// TIA Portal project "PKS_projektna_naloga_v1_9" (V15.1)

(* hardware
DEVICE "S7-1200 station_1"  S7-1200 Station
   slot 0: "Rack_0"  S7-1200 Rack  Rack  V1.0
   slot 1: "PLC_1"  CPU 1214C DC/DC/DC  6ES7 214-1AG40-0XB0  V4.2
DEVICE "HMI_1"  TP700 Comfort
   slot 0: "HMI_1"  TP700 Comfort  6AV2 124-0GC01-0AX0  15.1.0.0
   slot 1: "HMI_RT_1"  TP700 Comfort  6AV2 124-0GC01-0AX0  15.1.0.0
   slot 5: "HMI_1.IE_CP_1"  PROFINET Interface  15.0.1.0
      slot 1: "PROFINET Interface_1"  PROFINET Interface
         slot 1: "Port_1"  Port
         slot 2: "Port_2"  Port
   slot 7: "HMI_1.MPI/DP_CP_1"  MPI/DP Interface  15.0.1.0
*)

// ===== PLC "PLC_1"  CPU 1214C DC/DC/DC =====
// protected blocks, not shown: "FB_sim_model"

VAR_GLOBAL   // PLC tag table "Default tag table"
   "Tag_1" AT %MD0 : Time;
   "Tag_2" AT %M0.0 : Bool;
END_VAR

DATA_BLOCK "DB_podatki_procesa"   // DB2
{ S7_Optimized_Access := 'TRUE' }
VERSION : 0.1
   VAR
      V_žel : Real := 3000.0;   // želeni volumen v posodi v ml
      mr_AB_žel : Real := 0.35;   // želeno mešalno razmerje (mA : mB)
      ventil_A_pretok_max : Real := 200.0;   // max pretok ventila v ml/s
      ventil_B_pretok : Real := 200.0;   // pretok ventila B v g/s
      m_posode : Real := 200.0;   // masa (prazne) posode v g
      čas_prekinitve : Real := 0.1;   // čas prekinitve v s
      t_žel_meš : Real := 10.0;   // želeni čas postopka mešanja v s
      t_žel_vib : Real := 5.0;   // želeni čas postopka na vibracijski plošči v s
   END_VAR
   VAR RETAIN
      init_pogoj : Bool;   // pogoj za inicializacijo spremenljivk
   END_VAR
BEGIN
END_DATA_BLOCK

DATA_BLOCK "DB_spremenljivke"   // DB3
{ S7_Optimized_Access := 'TRUE' }
VERSION : 0.1
   VAR
      glavno_stikalo : Bool;   // glavno stikalo
      zasilni_izklop : Bool;   // tipka zasilni izklop
      reset : Bool;   // tipka reset
      tipka_stop : Bool;
      tipka_start : Bool;   // tipka start avtomatičnega procesa
      tipka_P_desno : Bool;   // tipka vklop podajalnika P desno
      tipka_P_levo : Bool;   // tipka vklop podajalnika P levo
      tipka_trak : Bool;   // tipka vklop traku "vklop ali izklop"
      dodaj_novo_paleto : Bool;
      odstrani_paleto : Bool;
      postavi_novo_posodo : Bool;
      premik_dozirnika_A_levo_desno : Bool;
      premik_dozirnika_B_levo_desno : Bool;
      pod_mesalo_dol : Bool;
      pod_mesalo_gor : Bool;
      "ventil_A+" : Bool;
      "ventil_A-" : Bool;
      vklop_izklop_ventila_B : Bool;
      vklopi_izklopi_mesalo : Bool;
      vklopi_izklopi_trak : Bool;
      vklop_izklop_VIB_plosce : Bool;
      vib_plošča_frek : Bool;
      rezim_rocno : Bool := 1;
      rezim_avtomaticno : Bool := 0;
      hitrost_traku : Bool := 0;   // 0 = slow, 1 FAST
      indikacija_avtomaticno : Bool := 0;
      indikacija_rocno : Bool := 0;
   END_VAR
BEGIN
END_DATA_BLOCK

DATA_BLOCK "DB_izhodne_spremenljivke"   // DB4
{ S7_Optimized_Access := 'TRUE' }
VERSION : 0.1
   VAR
      Pripravljenost : Bool;   // pripralvljenost
      Podajalnik_gre_LEVO : Bool;   // PPL
      Presezena_Limita_P_LEVO : Bool;   // S1
      Maks_Dovoljena_Lega_P_LEVO : Bool;   // S2
      Podajalnik_gre_DESNO : Bool;   // PPD
      Podajalnik_na_tehtnici : Bool;   // S3
      Maks_Dovoljena_Lega_P_DESNO : Bool;   // S4, tudi lega zacetka traka
      Presezena_Limita_P_DESNO : Bool;   // S5
      Tekoci_trak_VKLOPLJEN : Bool;   // MT
      Vib_Plata_Vklopljena : Bool;   // VP
      Posoda_na_plosci_LEVO : Bool;   // S6
      Posoda_na_plosci_DESNO : Bool;   // S7
      Posoda_v_koncni_legi_DESNO : Bool;   // S8
      Doz_A_LEVO : Bool;   // S9
      Doz_A_DESNO : Bool;   // S10
      Doz_B_LEVO : Bool;   // S11
      Doz_B_DESNO : Bool;   // S12
      Vklopljen_SPUST_MESALNIKA : Bool;   // PMD
      Vklopljen_DVIG_MESALNIKA : Bool;   // PMG
      Vklopljen_MESALNIK : Bool;   // MM -Mesalnik_se_vrti
      Maks_Dovoljena_Lega_MESALNIKA_GOR : Bool;   // S13
      Maks_Dovoljena_Lega_MESALNIKA_DOL : Bool;   // S14
      Ventil_A_DEG : Real;   // VA_stopinje
      Ventil_B_STANJE_ON_OFF : Bool;   // VB
      Volumen_DEJANSKI : Real;   // V_dej
      Skupna_masa : Real;   // masa
      Mesalno_razmerje_AB_dej : Real;   // mr_AB_dej
      Volumen_polite_mase : Real;   // V_polit
      Abs_ERROR : Real;   // ABSE
      Koda_napake : Word;   // error_word
      I_mesalo : Real;   // I_M
      U_mesalo : Real;   // U_M
      I_vib_plosce : Real;   // I_VP
      U_vib_plosce : Real;   // U_VP
   END_VAR
BEGIN
END_DATA_BLOCK

DATA_BLOCK "DB_vhodne_aktuatorjev"   // DB5
{ S7_Optimized_Access := 'TRUE' }
VERSION : 0.1
   VAR
      GLAVNO_STIKALO : Bool;
      ZASILNI_IZKLOP : Bool;
      RESET : Bool;
      TIPKA_START : Bool;
      PREMAKNI_POD_DESNO : Bool;
      PREMAKNI_POD_LEVO : Bool;
      TEKOCI_TRAK_ON_OFF : Bool;
      DODAJ_NOVO_PALETO : Bool;
      ODSTRANI_PALETO : Bool;
      POSTAVI_POSODO : Bool;
      PREMAKNI_DOZ_A_L_D : Bool;
      PREMAKNI_DOZ_B_L_D : Bool;
      MESALO_DOL : Bool;
      MESALO_GOR : Bool;
      "VENTIL_A_+" : Bool;
      "VENTIL_A_-" : Bool;
      VENTIL_B_ON_OFF : Bool;
      MESALO_ON_OFF : Bool;
      VIB_PLATA_ON_OFF : Bool;
      VIB_PLATA_FREQ : Bool;
      REZIM_ROCNO : Bool := 1;
      REZIM_AVTOMATICNO : Bool := 0;
      HITROST_TRAKU : Bool := 0;
   END_VAR
BEGIN
END_DATA_BLOCK

DATA_BLOCK "IZBERI_REZIM_DB"   // DB6
{ S7_Optimized_Access := 'TRUE' }
VERSION : 0.1
// stored: InstanceOfName IZBERI_REZIM
"IZBERI_REZIM"
BEGIN
END_DATA_BLOCK

DATA_BLOCK "Izracun_Energije_DB"   // DB7
{ S7_Optimized_Access := 'TRUE' }
VERSION : 0.1
// stored: InstanceOfName Izracun_Energije
"Izracun_Energije"
BEGIN
END_DATA_BLOCK

DATA_BLOCK "CHAT_GPT_ROCNO_DB"   // DB8
{ S7_Optimized_Access := 'TRUE' }
VERSION : 0.1
// stored: InstanceOfName CHAT_GPT_ROCNO
"CHAT_GPT_ROCNO"
BEGIN
END_DATA_BLOCK

DATA_BLOCK "DB_REZIM_AVTOMATSKO"   // DB10
{ S7_Optimized_Access := 'TRUE' }
VERSION : 0.1
// stored: InstanceOfName rezim_avtomatsko
"rezim_avtomatsko"
BEGIN
END_DATA_BLOCK

DATA_BLOCK "GLOBAL_Sync_Flags"   // DB12
{ S7_Optimized_Access := 'TRUE' }
VERSION : 0.1
   VAR
      Cmd_DodajPaleto_Req : Bool;
      Cmd_DodajPaleto_Ack : Bool;
      Cmd_DodajPosodo_Req : Bool;
      Cmd_DodajPosodo_Ack : Bool;
      Cmd_OdstraniPaleto_Req : Bool;
      Cmd_OdstraniPaleto_Ack : Bool;
      Preklopi_Na_Rocno : Bool;
   END_VAR
BEGIN
END_DATA_BLOCK

// folder: System blocks/Program resources

DATA_BLOCK "TIMER_RESET_150MS_DB"   // DB9
{ S7_Optimized_Access := 'TRUE' }
AUTHOR : Simatic
FAMILY : IEC
NAME : IEC_TMR
VERSION : 1.0
// stored: InstanceOfName IEC_TIMER
"IEC_TIMER"
BEGIN
END_DATA_BLOCK

DATA_BLOCK "TIMER_RESET_150MS_IZBERI_REZIM_DB"   // DB11
{ S7_Optimized_Access := 'TRUE' }
AUTHOR : Simatic
FAMILY : IEC
NAME : IEC_TMR
VERSION : 1.0
// stored: InstanceOfName IEC_TIMER
"IEC_TIMER"
BEGIN
END_DATA_BLOCK

DATA_BLOCK "Mesalnik_Cas_Mesanja_TON"   // DB13
{ S7_Optimized_Access := 'TRUE' }
AUTHOR : Simatic
FAMILY : IEC
NAME : IEC_TMR
VERSION : 1.0
// stored: InstanceOfName IEC_TIMER
"IEC_TIMER"
BEGIN
END_DATA_BLOCK

DATA_BLOCK "TIMER_Pocakaj_posoda_na_paleti_TON"   // DB14
{ S7_Optimized_Access := 'TRUE' }
AUTHOR : Simatic
FAMILY : IEC
NAME : IEC_TMR
VERSION : 1.0
// stored: InstanceOfName IEC_TIMER
"IEC_TIMER"
BEGIN
END_DATA_BLOCK

// folder: (top level)

FUNCTION_BLOCK "IZBERI_REZIM"   // FB2, SCL
{ S7_Optimized_Access := 'TRUE' }
VERSION : 0.1
   VAR
      Aktiven_Rezim_Avtomaticno : Bool;
      previous_reset : Bool;
      previous_rezim_avtomatsko : Bool;
      previous_rezim_rocno : Bool;
   END_VAR
   VAR_TEMP
      risingEdge_Reset : Bool;
      risingEdge_rezimRocno : Bool;
      risingEdge_rezimAvtomaticno : Bool;
      risingEdge_tipkaSTOP : Bool;
   END_VAR
   VAR CONSTANT
      Timer_const : Time := T#150ms;
   END_VAR
BEGIN
   // =======================================================================
   // BEGIN FB IZBERI REZIM
   // =======================================================================

   #risingEdge_Reset := "DB_spremenljivke".reset AND NOT #previous_reset;
   #risingEdge_rezimAvtomaticno := "DB_spremenljivke".rezim_avtomaticno AND NOT #previous_rezim_avtomatsko;
   #risingEdge_rezimRocno := "DB_spremenljivke".rezim_rocno AND NOT #previous_rezim_rocno;

   // 2. Reset Logic Handling

   "TIMER_RESET_150MS_IZBERI_REZIM_DB".TP(IN := #risingEdge_Reset,
                                          PT := #Timer_const,
                                          Q => "DB_vhodne_aktuatorjev".RESET);

   IF #risingEdge_Reset THEN
       #Aktiven_Rezim_Avtomaticno := FALSE;
   END_IF;

   // 3. Mode Selection Logic (as designed before)
   // --- Conditions to switch TO Automatic ---
   IF NOT #Aktiven_Rezim_Avtomaticno AND #risingEdge_rezimAvtomaticno THEN
       IF "DB_izhodne_spremenljivke".Pripravljenost THEN
           #Aktiven_Rezim_Avtomaticno := TRUE;
       END_IF;
   END_IF;

   IF "GLOBAL_Sync_Flags".Preklopi_Na_Rocno THEN
       #Aktiven_Rezim_Avtomaticno := FALSE;
       "GLOBAL_Sync_Flags".Preklopi_Na_Rocno:= FALSE;
   END_IF;


   IF #Aktiven_Rezim_Avtomaticno THEN
       "DB_vhodne_aktuatorjev".REZIM_AVTOMATICNO := TRUE;
       "DB_vhodne_aktuatorjev".REZIM_ROCNO := FALSE;
       "DB_REZIM_AVTOMATSKO"();

   ELSE
       "DB_vhodne_aktuatorjev".REZIM_AVTOMATICNO := FALSE;
       "DB_vhodne_aktuatorjev".REZIM_ROCNO := TRUE;
       "CHAT_GPT_ROCNO_DB"();
       "DB_vhodne_aktuatorjev".TIPKA_START := FALSE;
   END_IF;


   "DB_spremenljivke".indikacija_avtomaticno := #Aktiven_Rezim_Avtomaticno;
   "DB_spremenljivke".indikacija_rocno := NOT #Aktiven_Rezim_Avtomaticno;


   #previous_reset := "DB_spremenljivke".reset;
   #previous_rezim_avtomatsko := "DB_spremenljivke".rezim_avtomaticno;
   #previous_rezim_rocno := "DB_spremenljivke".rezim_rocno;
   // =======================================================================
   // END FB IZBERI REZIM
   // =======================================================================
END_FUNCTION_BLOCK

FUNCTION_BLOCK "rezim_avtomatsko"   // FB3, SCL
{ S7_Optimized_Access := 'TRUE' }
VERSION : 0.1
   VAR
      prev_START : Bool;
      prev_STOP : Bool;
      STANJE : Int;
      Stevilo_posod_na_paleti : Int;
      Stop_Tipka_Flag : Bool;
      Proces_Dokoncan_Flag : Bool;
      Masa_Grad_Mase_B_g : Real;
      Volumen_Vode_A_ml : Real;
      Timer_VENTIL_B_S : Int;
      prev_STANJE : Int := -1;
      Potreben_Vib_Time : Time;
      CAS_DozirnikaB_ON : Time;
      Izhod_MesalnikTimerja : Bool;
      Dokoncaj_Sekvenco_po_pritisku_stop : Bool;
   END_VAR
   VAR_TEMP
      risingEdge_START : Bool;
      risingEdge_STOP : Bool;
   END_VAR
   VAR CONSTANT
      Rho_Gradbene_Mase : Real := 1.7;   // kg/dm3
   END_VAR
BEGIN
   // =======================================================================
   // ZACETEK FUNKCIJSKEGA BLOKA // BEGIN FB rezim_avtomatsko
   // =======================================================================

   // =======================================================================
   // Rising Edge Detection for Start and Stop (Handled within this FB)
   // =======================================================================
   #risingEdge_START := "DB_spremenljivke".tipka_start AND NOT #prev_START;
   #risingEdge_STOP := "DB_spremenljivke".tipka_stop AND NOT #prev_STOP;
   // =======================================================================
   // Stop Button Handling (Request to stop sequence)
   // =======================================================================
   // Set Stop_Tipka_Flag on rising edge of Stop button if NOT already in a stop/error state
   IF #risingEdge_STOP AND (#STANJE > 0 AND #STANJE < 998) THEN // Assuming 998/999 are stop/error states
       #Stop_Tipka_Flag := TRUE;
       IF #STANJE >= 20 AND #STANJE <= 155 THEN
           #Dokoncaj_Sekvenco_po_pritisku_stop := TRUE; // Flag to complete current container sequence
       ELSE
           #Dokoncaj_Sekvenco_po_pritisku_stop := FALSE;
           #STANJE := 998; // Transition to immediate stop state
       END_IF;
   END_IF;

   // =======================================================================
   // Actuator Output Control (Controlled by state logic and sync flags/ack)
   // =======================================================================
   // Pulsed commands are handled by the OB30 logic reading the sync request flags.
   // Other actuator commands are set within the CASE statement.
   // It's good practice to explicitly set outputs to FALSE if they are not actively commanded TRUE in the current state.
   // Or, rely on the CASE statement setting outputs and have error/stop states turn them all off.

   // =======================================================================
   // Automatic Mode State Machine
   // =======================================================================

   CASE #STANJE OF
       0: // Idle - CAKAM NA START
           #Dokoncaj_Sekvenco_po_pritisku_stop := FALSE;
           #Stevilo_posod_na_paleti := 0;

           // Reset sinhronizacijskih flagov
           "GLOBAL_Sync_Flags".Cmd_DodajPaleto_Req := FALSE;
           "GLOBAL_Sync_Flags".Cmd_DodajPaleto_Ack := FALSE;
           "GLOBAL_Sync_Flags".Cmd_DodajPosodo_Req := FALSE;
           "GLOBAL_Sync_Flags".Cmd_DodajPosodo_Ack := FALSE;
           "GLOBAL_Sync_Flags".Cmd_OdstraniPaleto_Ack := FALSE;
           "GLOBAL_Sync_Flags".Cmd_OdstraniPaleto_Req := FALSE;

           #Volumen_Vode_A_ml := 0.0;
           #Masa_Grad_Mase_B_g := 0.0;
           #Potreben_Vib_Time := T#0ms;

           "DB_vhodne_aktuatorjev".PREMAKNI_POD_DESNO := FALSE;
           "DB_vhodne_aktuatorjev".PREMAKNI_POD_LEVO := FALSE;
           "DB_vhodne_aktuatorjev".PREMAKNI_DOZ_A_L_D := FALSE; // Or set to Left home state if needed
           "DB_vhodne_aktuatorjev".PREMAKNI_DOZ_B_L_D := FALSE; // Or set to Left home state if needed
           "DB_vhodne_aktuatorjev".MESALO_DOL := FALSE;
           "DB_vhodne_aktuatorjev".MESALO_GOR := FALSE;
           "DB_vhodne_aktuatorjev"."VENTIL_A_+" := FALSE;
           "DB_vhodne_aktuatorjev"."VENTIL_A_-" := FALSE;
           "DB_vhodne_aktuatorjev".VENTIL_B_ON_OFF := FALSE;
           "DB_vhodne_aktuatorjev".MESALO_ON_OFF := FALSE;
           "DB_vhodne_aktuatorjev".TEKOCI_TRAK_ON_OFF := FALSE;
           "DB_vhodne_aktuatorjev".VIB_PLATA_ON_OFF := FALSE;
           "DB_vhodne_aktuatorjev".HITROST_TRAKU := FALSE;
           "DB_vhodne_aktuatorjev".VIB_PLATA_FREQ := FALSE; // Set to safe state

           // Start button pressed AND System is Ready (Pripravljenost is checked in IZBERI_REZIM before calling this FB)
           IF #risingEdge_START THEN
               #STANJE := 10; // Transition to Cmd Add Pallet Request state
           END_IF;

           // Stop transition from Idle (Immediate Stop)
           IF #Stop_Tipka_Flag THEN
               #STANJE := 998; // Transition to stop state
           END_IF;


       10: // Cmd Add Pallet Request (in OB1)
           "GLOBAL_Sync_Flags".Cmd_DodajPaleto_Req := TRUE;
           // Reset the acknowledgement flag from a previous cycle if it was still set (safeguard)
           "GLOBAL_Sync_Flags".Cmd_DodajPaleto_Ack := FALSE;
           // Immediately transition to the waiting state
           #STANJE := 15; // Transition to Wait Pallet Ready
           // Poglej za stop (Immediate Stop)
           IF #Stop_Tipka_Flag THEN
               #STANJE := 998;
           END_IF;


       15: // Pocakaj da je paleta dodana (v OB30)
           // Wait for the acknowledgement flag from OB30 AND/OR process feedback
           IF "GLOBAL_Sync_Flags".Cmd_DodajPaleto_Ack THEN
               // Reset the acknowledgement flag as we've seen it
               "GLOBAL_Sync_Flags".Cmd_DodajPaleto_Ack := FALSE;
               #STANJE := 20;
           ELSE
               #STANJE := 15; // Stay in State 15 until Ack flag is set by OB30
           END_IF;

           // Check for stop request (Immediate Stop)
           IF #Stop_Tipka_Flag THEN
               #STANJE := 998;
           END_IF;


       20: // Cmd postavi posodo request (in OB30)
           "GLOBAL_Sync_Flags".Cmd_DodajPosodo_Req := TRUE;
           "GLOBAL_Sync_Flags".Cmd_DodajPosodo_Ack := FALSE;

           // Immediately transition to the waiting state
           #STANJE := 25; // Transition to Wait Container on P Home


       25: // Pocakaj sinhronizacijo (in OB30)
           IF "GLOBAL_Sync_Flags".Cmd_DodajPosodo_Ack THEN
               // Reset ack flag
               "GLOBAL_Sync_Flags".Cmd_DodajPosodo_Ack := FALSE;
               #STANJE := 30;
           ELSE
               #STANJE := 25;
           END_IF; // Stay in State 25 until Ack flag is set by OB30 and timeout elapses.


       30: //Premakni podajalnik do tehtnice (S3)
           IF NOT "DB_izhodne_spremenljivke".Podajalnik_na_tehtnici THEN
               "DB_vhodne_aktuatorjev".PREMAKNI_POD_DESNO := TRUE;
           ELSE
               "DB_vhodne_aktuatorjev".PREMAKNI_POD_DESNO := FALSE;
               #STANJE := 40;
           END_IF;


       40: // Dosage Calculation
           IF "DB_podatki_procesa".mr_AB_žel >= 0.2 AND "DB_podatki_procesa".mr_AB_žel <= 0.5 THEN

               // Masa_Grad_Mase_B_g = Massa komponente B 
               // Volumen_Vode_A_ml = Volumen komponente A v ml? 

               #Masa_Grad_Mase_B_g := "DB_podatki_procesa".V_žel / ((1 / #Rho_Gradbene_Mase) + ("DB_podatki_procesa".mr_AB_žel)); // Original izracun, assuming kg for B
               #Volumen_Vode_A_ml := "DB_podatki_procesa".mr_AB_žel * #Masa_Grad_Mase_B_g; // Original izracun, assuming ml for A
               #STANJE := 45; //Pojdi v naslednje stanje.

           ELSE
               #STANJE := 40;
           END_IF;


       45: // Cmd premakni dozirnik A desno
           IF "DB_izhodne_spremenljivke".Doz_A_LEVO THEN // Preveri da je trenutno levo
               "DB_vhodne_aktuatorjev".PREMAKNI_DOZ_A_L_D := TRUE; // Command Dispenser A Right (Set HIGH)
           ELSE
               IF "DB_izhodne_spremenljivke".Doz_A_DESNO THEN
                   #STANJE := 50; // Transition directly
               END_IF;
           END_IF;


       50: // Fill Component A (Water)
           #STANJE := 60;
           // "DB_vhodne_aktuatorjev".VENTIL_B_ON_OFF := FALSE;
           // IF "DB_izhodne_spremenljivke".Doz_A_DESNO AND "DB_izhodne_spremenljivke".Doz_B_LEVO AND "DB_izhodne_spremenljivke".Volumen_DEJANSKI <  (3000 * 0.33)THEN
           //     "DB_vhodne_aktuatorjev"."VENTIL_A_+" := TRUE;
           //     "DB_vhodne_aktuatorjev"."VENTIL_A_-" := FALSE;
           // END_IF;

           // IF "DB_izhodne_spremenljivke".Volumen_DEJANSKI >  (3000 * 0.65) THEN // Pulse or regulate near target
           //     // Implement proportional control or pulsing Valve A
           //     "DB_vhodne_aktuatorjev"."VENTIL_A_+" := FALSE; // Simple ON near target (Needs refinement)
           //     "DB_vhodne_aktuatorjev"."VENTIL_A_-" := TRUE;
           // END_IF;
           // // Transition from FILLING state happens *after* commanding close and waiting for confirmation.
           // IF "DB_izhodne_spremenljivke".Ventil_A_DEG = 0.0 THEN
           //     "DB_vhodne_aktuatorjev"."VENTIL_A_-" := FALSE;
           //     #STANJE := 60;
           // END_IF;


       60: // Cmd Premakni dozirnik A levo
           IF "DB_izhodne_spremenljivke".Doz_A_DESNO THEN
               "DB_vhodne_aktuatorjev".PREMAKNI_DOZ_A_L_D := FALSE;
           END_IF;

           IF "DB_izhodne_spremenljivke".Doz_A_LEVO THEN
               #STANJE := 65; // Pojdi v naslednje stanje.
           END_IF;


       65: // Cmd Premakni dozirnik B desno
           IF "DB_izhodne_spremenljivke".Doz_B_LEVO AND "DB_izhodne_spremenljivke".Doz_A_LEVO THEN
               "DB_vhodne_aktuatorjev".PREMAKNI_DOZ_B_L_D := TRUE; // Premakni desno
           ELSE
               IF "DB_izhodne_spremenljivke".Doz_B_DESNO AND "DB_izhodne_spremenljivke".Doz_A_LEVO THEN
                   #STANJE := 70;
               END_IF;
           END_IF;



       70: // Fill Component B (Aggregate)
           "DB_vhodne_aktuatorjev"."VENTIL_A_+" := FALSE;
           "DB_vhodne_aktuatorjev"."VENTIL_A_-" := FALSE;

           IF "DB_izhodne_spremenljivke".Skupna_masa < ("DB_podatki_procesa".m_posode + #Volumen_Vode_A_ml + #Masa_Grad_Mase_B_g) THEN
               "DB_vhodne_aktuatorjev".VENTIL_B_ON_OFF := TRUE; // Command Valve B Open
           ELSE
               "DB_vhodne_aktuatorjev".VENTIL_B_ON_OFF := FALSE;
               IF NOT "DB_izhodne_spremenljivke".Ventil_B_STANJE_ON_OFF THEN
                   #STANJE := 80;
               END_IF;
           END_IF;



       80: // Premakni dozirnik B levo Potem ko si napolnil z Grad. maso.
           IF "DB_izhodne_spremenljivke".Doz_B_DESNO AND NOT "DB_izhodne_spremenljivke".Ventil_B_STANJE_ON_OFF THEN
               "DB_vhodne_aktuatorjev".PREMAKNI_DOZ_B_L_D := FALSE; // Command Dispenser B Left (Set LOW)
           ELSE
               IF "DB_izhodne_spremenljivke".Doz_B_LEVO THEN
                   #STANJE := 90; // Transition directly
               ELSE
                   #STANJE := 80;
               END_IF;
           END_IF;



       90: // Spusti MESALNIK
           IF NOT "DB_izhodne_spremenljivke".Vklopljen_MESALNIK AND "DB_izhodne_spremenljivke".Maks_Dovoljena_Lega_MESALNIKA_GOR THEN
               "DB_vhodne_aktuatorjev".MESALO_GOR := FALSE;
               "DB_vhodne_aktuatorjev".MESALO_DOL := TRUE;

           END_IF;

           IF "DB_izhodne_spremenljivke".Maks_Dovoljena_Lega_MESALNIKA_DOL THEN
               "DB_vhodne_aktuatorjev".MESALO_GOR := FALSE;
               "DB_vhodne_aktuatorjev".MESALO_DOL := FALSE;
               #STANJE := 100;
           END_IF;



       100: // Motor mesalnika ON 

           IF #prev_STANJE <> 100 THEN
               "DB_vhodne_aktuatorjev".MESALO_ON_OFF := TRUE;
               "Mesalnik_Cas_Mesanja_TON".TON(IN := TRUE,
                                              PT := INT_TO_TIME(REAL_TO_INT("DB_podatki_procesa".t_žel_meš * 1000)), // t_žel_meš je v sec. (Real), PT rabi ms #TIME
                                              Q => #Izhod_MesalnikTimerja);
               #prev_STANJE := #STANJE;
           END_IF;

           IF "Mesalnik_Cas_Mesanja_TON".Q THEN
               "DB_vhodne_aktuatorjev".MESALO_ON_OFF := FALSE; // Turn off Mixer Motor
               "Mesalnik_Cas_Mesanja_TON".TON(IN := FALSE,
                                              PT := INT_TO_TIME(REAL_TO_INT("DB_podatki_procesa".t_žel_meš * 1000)));
               #STANJE := 110; // Transition to the next state (Assuming 105 is the next state, e.g., Mixer Up)
           END_IF;


       110: // Cmd Premakni mesalnik GOR v izhodiscno lego 
           IF "DB_izhodne_spremenljivke".Maks_Dovoljena_Lega_MESALNIKA_DOL THEN
               "DB_vhodne_aktuatorjev".MESALO_GOR := TRUE;
               "DB_vhodne_aktuatorjev".MESALO_DOL := FALSE; // Ensure not moving down
           END_IF;

           IF "DB_izhodne_spremenljivke".Maks_Dovoljena_Lega_MESALNIKA_GOR THEN
               "DB_vhodne_aktuatorjev".MESALO_GOR := FALSE;
               "DB_vhodne_aktuatorjev".MESALO_DOL := FALSE;
               #STANJE := 120;
           END_IF;


       120: // Premakni podajalnik s posodo do tekocega traku(Po mesanju in dvigu mesalnika)

           IF "DB_izhodne_spremenljivke".Podajalnik_na_tehtnici THEN
               "DB_vhodne_aktuatorjev".PREMAKNI_POD_DESNO := TRUE;
               "DB_vhodne_aktuatorjev".PREMAKNI_POD_LEVO := FALSE;
           END_IF;

           IF "DB_izhodne_spremenljivke".Maks_Dovoljena_Lega_P_DESNO THEN
               "DB_vhodne_aktuatorjev".PREMAKNI_POD_DESNO := FALSE;
               "DB_vhodne_aktuatorjev".PREMAKNI_POD_LEVO := FALSE;
               #STANJE := 130;
           END_IF;


       130: // Prizigi tekoci trak in vib plosco
           IF "DB_izhodne_spremenljivke".Maks_Dovoljena_Lega_P_DESNO AND (#prev_STANJE <> 130) THEN // Ce je posoda na zacetku na podlagi mase izaracunaj zeljen cas vibracije

               "DB_vhodne_aktuatorjev".TEKOCI_TRAK_ON_OFF := TRUE;
               "DB_vhodne_aktuatorjev".HITROST_TRAKU := FALSE;

               #Potreben_Vib_Time := INT_TO_TIME(REAL_TO_INT("DB_podatki_procesa".t_žel_vib * 1000));// Default time (ms)

               IF "DB_izhodne_spremenljivke".Skupna_masa > 1500 THEN // Preveri maso
                   #Potreben_Vib_Time := INT_TO_TIME(REAL_TO_INT("DB_podatki_procesa".t_žel_vib * 2000)); // Podvoji time if mass > 1.5kg
               END_IF;

           END_IF;

           IF NOT "DB_izhodne_spremenljivke".Maks_Dovoljena_Lega_P_LEVO THEN
               "DB_vhodne_aktuatorjev".PREMAKNI_POD_LEVO := TRUE;
           ELSE
               "DB_vhodne_aktuatorjev".PREMAKNI_POD_LEVO := FALSE;
               "DB_vhodne_aktuatorjev".PREMAKNI_POD_DESNO := FALSE;
           END_IF;

           IF "DB_izhodne_spremenljivke".Posoda_na_plosci_LEVO THEN
               "DB_vhodne_aktuatorjev".VIB_PLATA_ON_OFF := TRUE;
           END_IF;

           IF "DB_izhodne_spremenljivke".Posoda_na_plosci_DESNO THEN
               "DB_vhodne_aktuatorjev".VIB_PLATA_ON_OFF := FALSE;
           END_IF;

           IF "DB_izhodne_spremenljivke".Posoda_v_koncni_legi_DESNO THEN
               #STANJE := 140;
           END_IF;


       140: // Posoda postavljena na konec palete / inc. st. posod na paleti
           IF #prev_STANJE <> 140 THEN
               #prev_STANJE := 140;
               "TIMER_Pocakaj_posoda_na_paleti_TON".TON(IN := TRUE,
                                                        PT := T#3000ms);
           END_IF;
           IF "TIMER_Pocakaj_posoda_na_paleti_TON".Q THEN

               "TIMER_Pocakaj_posoda_na_paleti_TON".TON(IN := FALSE,
                                                        PT := T#3000ms);

               "DB_vhodne_aktuatorjev".TEKOCI_TRAK_ON_OFF := FALSE;
               #Stevilo_posod_na_paleti := #Stevilo_posod_na_paleti + 1;
               #STANJE := 150; // tranzicija, preveri paleta polna

           END_IF;


       150: // Preveri ce je paleta polna in se odloci ali lahko dodas novo posodo
           IF #Stevilo_posod_na_paleti = 6 THEN // palleta polna
               #prev_STANJE := 150;
               #STANJE := 155; // STANJE ---> odstrani paleto
           ELSE
               #STANJE := 20; 
           END_IF;

           // Check for stop request (Immediate Stop)
           IF #Stop_Tipka_Flag THEN
               #STANJE := 998;
           END_IF;


       155: // paleta polna -> odstrani paleto request
           #Stevilo_posod_na_paleti := 0;
           IF #prev_STANJE <> 155 THEN
               "GLOBAL_Sync_Flags".Cmd_OdstraniPaleto_Req := TRUE;
               #prev_STANJE := 155;
           END_IF;

           IF "GLOBAL_Sync_Flags".Cmd_OdstraniPaleto_Ack THEN
               "GLOBAL_Sync_Flags".Cmd_OdstraniPaleto_Ack := FALSE;

               #STANJE := 0;
           END_IF;

           // Check for stop request (Immediate Stop)
           IF #Stop_Tipka_Flag THEN
               #STANJE := 998;
           END_IF;

       998: // Stop stanje ---> rocni nacin
           // izklopi vse aktuatorje
           "resetiraj_aktuatorje"();
           "GLOBAL_Sync_Flags".Preklopi_Na_Rocno := TRUE;
           // resetiraj flage ce slucajno se niso
           "GLOBAL_Sync_Flags".Cmd_DodajPaleto_Req := FALSE;
           "GLOBAL_Sync_Flags".Cmd_DodajPaleto_Ack := FALSE;
           "GLOBAL_Sync_Flags".Cmd_DodajPosodo_Req := FALSE;
           "GLOBAL_Sync_Flags".Cmd_DodajPosodo_Ack := FALSE;
           "GLOBAL_Sync_Flags".Cmd_OdstraniPaleto_Req := FALSE;
           "GLOBAL_Sync_Flags".Cmd_OdstraniPaleto_Ack := FALSE;

           #Stop_Tipka_Flag := FALSE;
           #prev_STANJE := 0;
           #STANJE := 0;

   END_CASE;
   // =======================================================================
   // Update Previous States for Edge Detection (within this FB)
   // =======================================================================
   #prev_START := "DB_spremenljivke".tipka_start;
   #prev_STOP := "DB_spremenljivke".tipka_stop;
   // =======================================================================
   // END OF FUNCTION BLOCK
   // =======================================================================
END_FUNCTION_BLOCK

FUNCTION_BLOCK "CHAT_GPT_ROCNO"   // FB4, SCL
{ S7_Optimized_Access := 'TRUE' }
VERSION : 0.1
   VAR
      prev_tipka_P_DESNO : Bool;
      prev_tipka_P_LEVO : Bool;
      prev_reset : Bool;
      prev_tipka_trak : Bool;
   END_VAR
   VAR_TEMP
      risingEdge_tipka_P_DESNO : Bool;
      risingEdge_tipka_P_LEVO : Bool;
      dovoli_P_DESNO : Bool;
      dovoli_P_LEVO : Bool;
      condition_Set_Right : Bool;
      condition_Reset_Right : Bool;
      condition_Set_Left : Bool;
      condition_Reset_Left : Bool;
      risingEdge_reset : Bool;
      allow_Mesalo_Dol : Bool;
      allow_Mesalo_Gor : Bool;
      allow_Ventil_A_Odpri : Bool;
      allow_Ventil_A_Zapri : Bool;
      allow_Ventil_B_Vklop : Bool;
      allow_Mesalo_Vklop : Bool;
      risingEdge_tipka_trak : Bool;
   END_VAR
   VAR CONSTANT
      Timer_150MS_Const : Time := T#150ms;
   END_VAR
BEGIN

   // =======================================================================
   // 0. Detekcija pozitivne fronte za HMI ukaze
   // =======================================================================
   // Izračunamo edge_triggerje PRED glavno logiko, shranimo v TEMP spremenljivke.
   // Stanje 'prev_' se posodobi na KONCU bloka.

   #risingEdge_tipka_P_DESNO := "DB_spremenljivke".tipka_P_desno AND NOT #prev_tipka_P_DESNO;
   #risingEdge_tipka_P_LEVO := "DB_spremenljivke".tipka_P_levo AND NOT #prev_tipka_P_LEVO;
   #risingEdge_reset := "DB_spremenljivke".reset AND NOT #prev_reset;
   #risingEdge_tipka_trak := "DB_spremenljivke".vklopi_izklopi_trak AND NOT #prev_tipka_trak;
   // // =======================================================================
   // // 0. Reset, generiraj 150ms dolg pulz na "DB_vhodne_aktuatorjev".RESET ko se zgodi risingEdge na tipki reset
   // // =======================================================================

   REGION RESET
       "TIMER_RESET_150MS_DB".TP(IN:=#risingEdge_reset,
                                 PT:=#Timer_150MS_Const,
                                 Q=>"DB_vhodne_aktuatorjev".RESET);
       IF "TIMER_RESET_150MS_DB".Q THEN
           "resetiraj_aktuatorje"(); // TOOD potrebno je tudi resetirat procesne spremenljivke
       END_IF;

   END_REGION
   // // =======================================================================
   // // 1. Osnovni ukazi (Dodaj/Odstrani paleto, Nova posoda)
   // // =======================================================================

   REGION Dodajanje in odstranjevanje palete/posode

       IF ("DB_spremenljivke".dodaj_novo_paleto) THEN
           "DB_vhodne_aktuatorjev".ODSTRANI_PALETO := FALSE;
           "DB_vhodne_aktuatorjev".DODAJ_NOVO_PALETO := TRUE;
       ELSE
           "DB_vhodne_aktuatorjev".DODAJ_NOVO_PALETO := FALSE;
       END_IF;
       IF ("DB_spremenljivke".odstrani_paleto) THEN
           "DB_vhodne_aktuatorjev".ODSTRANI_PALETO := TRUE;
           "DB_vhodne_aktuatorjev".DODAJ_NOVO_PALETO := FALSE;
       END_IF;
       IF ("DB_spremenljivke".postavi_novo_posodo) THEN
           "DB_vhodne_aktuatorjev".POSTAVI_POSODO :=TRUE;
       ELSE
           "DB_vhodne_aktuatorjev".POSTAVI_POSODO := FALSE;
       END_IF;

   END_REGION 


   // =======================================================================
   // 2. KRMILJENJE PODAJALNIKA P (P)
   // =======================================================================
   REGION Podajalnik_P_Control
       // --- Control for Feeder P Movement ---
       // Use rising edge of HMI buttons to initiate movement, subject to interlocks and strict mutual exclusion.
       // Movement stops immediately if opposite button is pressed or interlocks are broken.

       // First check if either button is pressed to STOP current movement
       IF #risingEdge_tipka_P_LEVO AND "DB_vhodne_aktuatorjev".PREMAKNI_POD_DESNO THEN
           // If left button pressed while moving right, just stop
           "DB_vhodne_aktuatorjev".PREMAKNI_POD_DESNO := FALSE;
       ELSIF #risingEdge_tipka_P_DESNO AND "DB_vhodne_aktuatorjev".PREMAKNI_POD_LEVO THEN
           // If right button pressed while moving left, just stop
           "DB_vhodne_aktuatorjev".PREMAKNI_POD_LEVO := FALSE;
       ELSE
           // Normal control logic when no opposite movement is happening

           // Latch the command to move Right based on rising edge and interlocks.
           IF NOT (
               "DB_izhodne_spremenljivke".Maks_Dovoljena_Lega_MESALNIKA_GOR AND
               "DB_izhodne_spremenljivke".Doz_A_LEVO AND
               "DB_izhodne_spremenljivke".Doz_B_LEVO AND
               NOT "DB_izhodne_spremenljivke".Maks_Dovoljena_Lega_P_DESNO
               ) THEN // Interlocks broken for Right
               "DB_vhodne_aktuatorjev".PREMAKNI_POD_DESNO := FALSE; // Reset Right command
           ELSIF #risingEdge_tipka_P_DESNO AND // Set Right command on rising edge
               "DB_izhodne_spremenljivke".Maks_Dovoljena_Lega_MESALNIKA_GOR AND
               "DB_izhodne_spremenljivke".Doz_A_LEVO AND
               "DB_izhodne_spremenljivke".Doz_B_LEVO AND
               NOT "DB_izhodne_spremenljivke".Maks_Dovoljena_Lega_P_DESNO AND
               NOT "DB_vhodne_aktuatorjev".PREMAKNI_POD_LEVO THEN // ONLY set if Left is NOT active
               "DB_vhodne_aktuatorjev".PREMAKNI_POD_DESNO := TRUE;
           END_IF;

           // Latch the command to move Left based on rising edge and interlocks.
           IF NOT (
               "DB_izhodne_spremenljivke".Maks_Dovoljena_Lega_MESALNIKA_GOR AND
               "DB_izhodne_spremenljivke".Doz_A_LEVO AND
               "DB_izhodne_spremenljivke".Doz_B_LEVO AND
               NOT "DB_izhodne_spremenljivke".Maks_Dovoljena_Lega_P_LEVO
               ) THEN // Interlocks broken for Left
               "DB_vhodne_aktuatorjev".PREMAKNI_POD_LEVO := FALSE; // Reset Left command
           ELSIF #risingEdge_tipka_P_LEVO AND // Set Left command on rising edge
               "DB_izhodne_spremenljivke".Maks_Dovoljena_Lega_MESALNIKA_GOR AND
               "DB_izhodne_spremenljivke".Doz_A_LEVO AND
               "DB_izhodne_spremenljivke".Doz_B_LEVO AND
               NOT "DB_izhodne_spremenljivke".Maks_Dovoljena_Lega_P_LEVO AND
               NOT "DB_vhodne_aktuatorjev".PREMAKNI_POD_DESNO THEN // ONLY set if Right is NOT active
               "DB_vhodne_aktuatorjev".PREMAKNI_POD_LEVO := TRUE;
           END_IF;
       END_IF;

       // Final safeguard - should not be necessary with above logic, but good practice.
       // If somehow both are active, turn both off.
       IF "DB_vhodne_aktuatorjev".PREMAKNI_POD_DESNO AND "DB_vhodne_aktuatorjev".PREMAKNI_POD_LEVO THEN
           "DB_vhodne_aktuatorjev".PREMAKNI_POD_DESNO := FALSE;
           "DB_vhodne_aktuatorjev".PREMAKNI_POD_LEVO := FALSE;
       END_IF;

   END_REGION // Podajalnik_P_Control

   // =======================================================================
   // 3. Krmiljenje dozirnikov (M)
   // =======================================================================
   REGION Dozirnik_A_Control
       IF "DB_izhodne_spremenljivke".Maks_Dovoljena_Lega_MESALNIKA_GOR AND NOT "DB_izhodne_spremenljivke".Vklopljen_DVIG_MESALNIKA AND NOT "DB_izhodne_spremenljivke".Vklopljen_SPUST_MESALNIKA AND NOT "DB_izhodne_spremenljivke".Vklopljen_MESALNIK THEN
           "DB_vhodne_aktuatorjev".PREMAKNI_DOZ_A_L_D := "DB_spremenljivke".premik_dozirnika_A_levo_desno;
       END_IF;
   END_REGION // Dozirnik_B_Control

   REGION Dozirnik_B_Control
       // --- Control for Dispenser B Position (Latched by Toggle Button with Interlocks) ---
       // Toggle the state of the actuator input on the rising edge of the HMI button, if interlocks are met.
       // Assuming PREMAKNI_DOZ_B_L_D HIGH commands one position, LOW commands the other.

       // Interlock condition to allow toggling for Dispenser B:
       // Mixer must be up AND (Dispenser B is in Left position OR Dispenser B is in Right position)
       IF "DB_izhodne_spremenljivke".Maks_Dovoljena_Lega_MESALNIKA_GOR AND NOT "DB_izhodne_spremenljivke".Vklopljen_DVIG_MESALNIKA AND NOT "DB_izhodne_spremenljivke".Vklopljen_SPUST_MESALNIKA AND NOT "DB_izhodne_spremenljivke".Vklopljen_MESALNIK THEN
           "DB_vhodne_aktuatorjev".PREMAKNI_DOZ_B_L_D := "DB_spremenljivke".premik_dozirnika_B_levo_desno;
       END_IF;

   END_REGION // Dozirnik_B_Control

   // =======================================================================
   // 4. KRMILJENJE PODAJALNIKA MEŠALA (M)
   // =======================================================================
   REGION Podajalnik_Mesala_Control

       // Conditions for moving Down
       #allow_Mesalo_Dol := "DB_spremenljivke".pod_mesalo_dol AND // HMI command (Momentary)
       NOT "DB_izhodne_spremenljivke".Vklopljen_MESALNIK AND // Mixer motor must be off
       "DB_izhodne_spremenljivke".Podajalnik_na_tehtnici AND // ali lahko damo mesalo dol tudi ce ni posoda na tehtnici/
       "DB_izhodne_spremenljivke".Doz_A_LEVO AND
       "DB_izhodne_spremenljivke".Doz_B_LEVO AND
       NOT "DB_spremenljivke".pod_mesalo_gor AND
       NOT "DB_izhodne_spremenljivke".Maks_Dovoljena_Lega_MESALNIKA_DOL; // Prevent simultaneous command from HMI

       // Conditions for moving Up
       #allow_Mesalo_Gor := "DB_spremenljivke".pod_mesalo_gor AND // HMI command (Momentary)
       "DB_izhodne_spremenljivke".Doz_A_LEVO AND
       "DB_izhodne_spremenljivke".Doz_B_LEVO AND
       NOT "DB_izhodne_spremenljivke".Vklopljen_MESALNIK AND // Mixer motor must be off
       NOT "DB_spremenljivke".pod_mesalo_dol AND
       NOT "DB_izhodne_spremenljivke".Maks_Dovoljena_Lega_MESALNIKA_GOR; // Prevent simultaneous command from HMI

       // --- Set outputs for FB1 ---
       // Direct assignment from allowed conditions (outputs will be ON as long as HMI button is pressed AND interlocks are met)
       "DB_vhodne_aktuatorjev".MESALO_DOL := #allow_Mesalo_Dol; // Input for moving down
       "DB_vhodne_aktuatorjev".MESALO_GOR := #allow_Mesalo_Gor; // Input for moving up

       // Note: If these inputs to the OB30 FB actually require a pulse or timed signal
       // for reliable triggering in the slower cycle, this direct assignment might
       // need to be replaced with a pulse timer logic similar to the Reset/Pallet commands
       // discussed previously.
   END_REGION // Podajalnik_Mesala_Control

   // =======================================================================
   // 6. KRMILJENJE VENTILA A
   // =======================================================================
   REGION Ventil_A_Control
       // --- Pogoji za odpiranje/zapiranje A (momentary tipke) ---
       #allow_Ventil_A_Odpri := "DB_spremenljivke"."ventil_A+" AND // HMI ukaz
       "DB_izhodne_spremenljivke".Doz_A_DESNO AND     // Dozirnik A mora biti desno
       "DB_izhodne_spremenljivke".Doz_B_LEVO AND  // Ventil B mora biti zaprt
       "DB_izhodne_spremenljivke".Maks_Dovoljena_Lega_MESALNIKA_GOR AND
       NOT "DB_spremenljivke"."ventil_A-"; // Ne zapiramo hkrati

       #allow_Ventil_A_Zapri := "DB_spremenljivke"."ventil_A-" AND // HMI ukaz
       NOT "DB_spremenljivke"."ventil_A+"; // Ne odpiramo hkrati

       // --- Nastavitev izhodov za FB1 ---
       "DB_vhodne_aktuatorjev"."VENTIL_A_+" := #allow_Ventil_A_Odpri;
       "DB_vhodne_aktuatorjev"."VENTIL_A_-" := #allow_Ventil_A_Zapri;

   END_REGION // Ventil_A_Control

   // =======================================================================
   // 7. KRMILJENJE VENTILA B (Toggle)
   // =======================================================================
   REGION Ventil_B_Control
       // --- Pogoji za vklop/izklop B ---
       #allow_Ventil_B_Vklop := "DB_spremenljivke".vklop_izklop_ventila_B AND            // Želeno stanje je VKLOP
       "DB_izhodne_spremenljivke".Doz_B_DESNO AND // Dozirnik B mora biti desno
       "DB_izhodne_spremenljivke".Doz_A_LEVO AND // Dozirnik A mora biti levo
       ("DB_izhodne_spremenljivke".Ventil_A_DEG = 0.0); // Ventil A mora biti zaprt

       // --- Nastavitev izhoda za FB1 ---
       // FB1 vhod 'ventil_B_V_I' pričakuje stalni signal za stanje.

       "DB_vhodne_aktuatorjev".VENTIL_B_ON_OFF := #allow_Ventil_B_Vklop;


   END_REGION // Ventil_B_Control

   // =======================================================================
   // 8. KRMILJENJE MOTORJA MEŠALA (Toggle)
   // =======================================================================
   REGION Mesalo_Motor_Control

       // --- Pogoji za vklop/izklop MM ---
       #allow_Mesalo_Vklop := "DB_spremenljivke".vklopi_izklopi_mesalo AND           // Želeno stanje VKLOP
       "DB_izhodne_spremenljivke".Maks_Dovoljena_Lega_MESALNIKA_DOL;    // Mešalo mora biti spodaj

       "DB_vhodne_aktuatorjev".MESALO_ON_OFF := #allow_Mesalo_Vklop;

   END_REGION // Mesalo_Motor_Control

   // =======================================================================
   // 9. KRMILJENJE TEKOČEGA TRAKU (Toggle)
   // =======================================================================
   REGION Trak_Control
       // Dokumentacija omenja DLF! (rising edge) za tipko_trak,
       // 'vklopi_izklopi_trak' v DB_spremenljivke nakazuje preklop.
       IF #risingEdge_tipka_trak THEN
           "DB_vhodne_aktuatorjev".TEKOCI_TRAK_ON_OFF := NOT "DB_vhodne_aktuatorjev".TEKOCI_TRAK_ON_OFF;
       END_IF;
       // Nastavitev hitrosti traku (FB1 vhod trak_hitrost je Bool)
       "DB_vhodne_aktuatorjev".HITROST_TRAKU := "DB_spremenljivke".hitrost_traku;

   END_REGION // Trak_Control

   // =======================================================================
   // 10. KRMILJENJE VIBRACIJSKE PLOŠČE (Toggle)
   // =======================================================================
   REGION Vib_Control
       // --- Pogoji za vklop/izklop Vib ---

       // Nastavitev frekvence (FB1 vhod vib_plošča_frek je Bool)
       "DB_vhodne_aktuatorjev".VIB_PLATA_ON_OFF := "DB_spremenljivke".vklop_izklop_VIB_plosce;

   END_REGION // Vib_Control


   // =======================================================================
   // 12. Posodabljanje prejšnjih stanj za detekcijo fronte
   // ===================================================== ==================
   // Mora bit na KONCU bloka, po vsej logiki, ki uporablja detekcijo front.

   #prev_reset := "DB_spremenljivke".reset;
   #prev_tipka_P_DESNO := "DB_spremenljivke".tipka_P_desno;
   #prev_tipka_P_LEVO := "DB_spremenljivke".tipka_P_levo;
   #prev_tipka_trak := "DB_spremenljivke".vklopi_izklopi_trak;
END_FUNCTION_BLOCK

FUNCTION_BLOCK "Izracun_Energije"   // FB5, SCL
{ S7_Optimized_Access := 'TRUE' }
VERSION : 0.1
   VAR
      Akumulirana_energija_mesala : Real;
      Akumulirana_energija_vib_plosce : Real;
   END_VAR
   VAR CONSTANT
      Cycle_Time : Time := T#100ms;
   END_VAR
BEGIN
   // Conceptual code to be placed within the OB30 execution cycle,
   // AFTER the call to FB_sim_model

   // Assume these are STATIC variables declared elsewhere in the OB30 context (e.g., in the calling FB's instance DB)
   // VAR_STATIC
   //    ENERGIJA ZA MESALNIK: Real := 0.0; // Use Real or LReal depending on expected energy range
   //    ENERGIJA ZA VIB. PLOSCO: Real := 0.0; // Use Real or LReal

   // CASOVNI INTERVAL 100ms (fixed at OB30 cycle time/ interrupt time) #Cycle_Time

   // Energy Calculation for Mixer
   // Only calculate energy when the mixer is actually running
   IF "DB_izhodne_spremenljivke".Vklopljen_MESALNIK THEN
       // Power (Watts) = Voltage (Volts) * Current (Amps)
       // Energy added (Joules) = Power (Watts) * Time (seconds)
       #Akumulirana_energija_mesala := #Akumulirana_energija_mesala + ("DB_izhodne_spremenljivke".U_mesalo * "DB_izhodne_spremenljivke".I_mesalo * INT_TO_REAL(TIME_TO_INT(#Cycle_Time)) / 1000.0) /1000; // U v VOLTIH, I v AMPERGIH, pretvorba ms v sec
   END_IF;

   // Energy Calculation for Vibration Plate
   // Only calculate energy when the vibration plate is actually running
   IF "DB_izhodne_spremenljivke".Vib_Plata_Vklopljena THEN
       // Power (Watts) = Voltage (Volts) * Current (Amps)
       // Energy added (Joules) = Power (Watts) * Time (seconds)
       #Akumulirana_energija_vib_plosce := #Akumulirana_energija_vib_plosce + ("DB_izhodne_spremenljivke".U_vib_plosce * "DB_izhodne_spremenljivke".I_vib_plosce * INT_TO_REAL(TIME_TO_INT(#Cycle_Time)) / 1000.0)/1000; //v kWh
   END_IF;

   //RESETIRAJ typically when the entire process is reset (e.g., based on the system reset signal).
   IF "DB_vhodne_aktuatorjev".RESET THEN // Or your main system reset condition
       #Akumulirana_energija_mesala := 0.0;
       #Akumulirana_energija_vib_plosce := 0.0;
   END_IF;
END_FUNCTION_BLOCK

FUNCTION "FC_init" : Void   // FC1, LAD
{ S7_Optimized_Access := 'TRUE' }
VERSION : 0.1
   VAR_OUTPUT
      tipka_levo : Bool;
      tipka_desno : Bool;
      tipka_trak : Bool;
      tipka_start : Bool;
   END_VAR
BEGIN

REGION Network 1
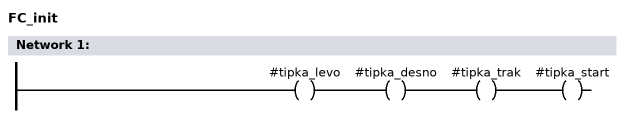
   RUNG wire#powerrail
      Coil( #tipka_levo )
      Coil( #tipka_desno )
      Coil( #tipka_trak )
      Coil( #tipka_start )
   END_RUNG
   // the same network as SCL:
   #tipka_levo := TRUE;
   #tipka_desno := TRUE;
   #tipka_trak := TRUE;
   #tipka_start := TRUE;
END_REGION
END_FUNCTION

FUNCTION "resetiraj_aktuatorje" : Void   // FC2, SCL
{ S7_Optimized_Access := 'TRUE' }
VERSION : 0.1
BEGIN
   // =======================================================================
   // 1. Initialization of Actuator Commands to FALSE
   // =======================================================================
   // Ensure that commands are active only when explicitly set by the logic.
   "DB_vhodne_aktuatorjev".PREMAKNI_POD_DESNO := FALSE; // Ime vhoda iz dokumentacije FB1
   "DB_vhodne_aktuatorjev".PREMAKNI_POD_LEVO := FALSE; // Ime vhoda iz dokumentacije FB1
   "DB_vhodne_aktuatorjev".PREMAKNI_DOZ_A_L_D := FALSE;// Ime vhoda iz dokumentacije FB1
   "DB_vhodne_aktuatorjev".PREMAKNI_DOZ_B_L_D := FALSE;// Ime vhoda iz dokumentacije FB1
   "DB_vhodne_aktuatorjev".MESALO_DOL := FALSE;// Ime vhoda iz dokumentacije FB1
   "DB_vhodne_aktuatorjev".MESALO_GOR := FALSE;// Ime vhoda iz dokumentacije FB1
   "DB_vhodne_aktuatorjev"."VENTIL_A_+" := FALSE;// Ime vhoda iz dokumentacije FB1
   "DB_vhodne_aktuatorjev"."VENTIL_A_-" := FALSE;// Ime vhoda iz dokumentacije FB1
   "DB_vhodne_aktuatorjev".VENTIL_B_ON_OFF := FALSE;// Ime vhoda iz dokumentacije FB1
   "DB_vhodne_aktuatorjev".MESALO_ON_OFF := FALSE;// Ime vhoda iz dokumentacije FB1 (meš_V_I ali mesalo_V_I?) - PREVERI IME!
   "DB_vhodne_aktuatorjev".TEKOCI_TRAK_ON_OFF := FALSE;// Ime vhoda iz dokumentacije FB1
   "DB_vhodne_aktuatorjev".VIB_PLATA_ON_OFF := FALSE;// Ime vhoda iz dokumentacije FB1
   "DB_vhodne_aktuatorjev".DODAJ_NOVO_PALETO := FALSE;// Ime vhoda iz dokumentacije FB1
   "DB_vhodne_aktuatorjev".ODSTRANI_PALETO := FALSE;// Ime vhoda iz dokumentacije FB1
   "DB_vhodne_aktuatorjev".POSTAVI_POSODO := FALSE;// Ime vhoda iz dokumentacije FB1
   // hitrost_traku in vib_plošča_frek se nastavita posebej
END_FUNCTION

FUNCTION "OB30_Network1" : Void   // FC3, SCL
{ S7_Optimized_Access := 'TRUE' }
VERSION : 0.1
BEGIN

   // Process Place Pallet Command Request
   IF "GLOBAL_Sync_Flags".Cmd_DodajPaleto_Req THEN
       "DB_vhodne_aktuatorjev".DODAJ_NOVO_PALETO := TRUE;
       "GLOBAL_Sync_Flags".Cmd_DodajPaleto_Req  := FALSE;
       "GLOBAL_Sync_Flags".Cmd_DodajPaleto_Ack := TRUE;
   // ELSE
   //     "DB_vhodne_aktuatorjev".DODAJ_NOVO_PALETO := FALSE;
   END_IF;

   // Process Place Container Command Request
   IF "GLOBAL_Sync_Flags".Cmd_DodajPosodo_Req THEN
       "DB_vhodne_aktuatorjev".POSTAVI_POSODO := TRUE;
       "GLOBAL_Sync_Flags".Cmd_DodajPosodo_Req:= FALSE;
       "GLOBAL_Sync_Flags".Cmd_DodajPosodo_Ack := TRUE;
   // ELSE
   //     "DB_vhodne_aktuatorjev".POSTAVI_POSODO := FALSE;
   END_IF;

   // Process Remove Pallet Command Request
   IF "GLOBAL_Sync_Flags".Cmd_OdstraniPaleto_Req THEN
       "DB_vhodne_aktuatorjev".ODSTRANI_PALETO := TRUE;
       "GLOBAL_Sync_Flags".Cmd_OdstraniPaleto_Req := FALSE;
       "GLOBAL_Sync_Flags".Cmd_OdstraniPaleto_Ack := TRUE;
   // ELSE
   //     "DB_vhodne_aktuatorjev".ODSTRANI_PALETO := FALSE;
   END_IF;
END_FUNCTION

FUNCTION "OB30_Network4" : Void   // FC4, SCL
{ S7_Optimized_Access := 'TRUE' }
VERSION : 0.1
BEGIN
       "DB_vhodne_aktuatorjev".DODAJ_NOVO_PALETO := FALSE;
       "DB_vhodne_aktuatorjev".POSTAVI_POSODO := FALSE;
       "DB_vhodne_aktuatorjev".ODSTRANI_PALETO := FALSE;
END_FUNCTION

ORGANIZATION_BLOCK "Main"   // OB1, SCL, ProgramCycle
TITLE = "Main Program Sweep (Cycle)"
{ S7_Optimized_Access := 'TRUE' }
VERSION : 0.1
   VAR_INPUT
      Initial_Call : Bool;   // Initial call of this OB
      Remanence : Bool;   // =True, if remanent data are available
   END_VAR
BEGIN
   // =======================================================================
   // BEGIN OB1
   // =======================================================================

   // *** CRITICAL SAFETY CHECK FIRST ***
   IF "DB_spremenljivke".zasilni_izklop OR NOT "DB_spremenljivke".glavno_stikalo THEN
   // --- HARD STOP LOGIC ---
    // Command FB1 E-Stop/Switch OFF inputs:
       "resetiraj_aktuatorje"();
       "DB_vhodne_aktuatorjev".ZASILNI_IZKLOP := TRUE; // Assume FB1 has E-Stop input
       "DB_vhodne_aktuatorjev".GLAVNO_STIKALO := FALSE; // Assume FB1 has Main Switch input

       RETURN; 
   END_IF;
   // --- NORMAL OPERATION LOGIC (Runs ONLY if NO Hard Stop) ---
   // Set FB1 inputs indicating normal operation state (only needed if NOT in hard stop)
   "DB_vhodne_aktuatorjev".ZASILNI_IZKLOP := "DB_spremenljivke".zasilni_izklop; // Reset E-Stop input to FB1
   "DB_vhodne_aktuatorjev".GLAVNO_STIKALO := "DB_spremenljivke".glavno_stikalo; // Set Main Switch input to FB1

   "IZBERI_REZIM_DB"(); // Call your mode selector FB

   // ====================================================
   // END OB1 
   // ====================================================
END_ORGANIZATION_BLOCK

ORGANIZATION_BLOCK "Cyclic interrupt"   // OB30, LAD, CyclicInterrupt
{ S7_Optimized_Access := 'TRUE' }
VERSION : 0.1
   VAR_INPUT
      Initial_Call : Bool;   // Initial call of this OB
      Event_Count : Int;   // Events discarded
   END_VAR
   VAR_TEMP
      cas : Time;
      stevec_casa : DInt;
   END_VAR
BEGIN

REGION Network 1
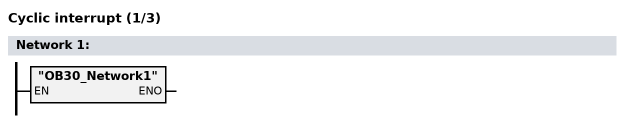
   RUNG wire#powerrail
      "OB30_Network1"()
   END_RUNG
   // the same network as SCL:
   "OB30_Network1"();
END_REGION

REGION Network 2: Simulacijski model
   // V tem networku je model
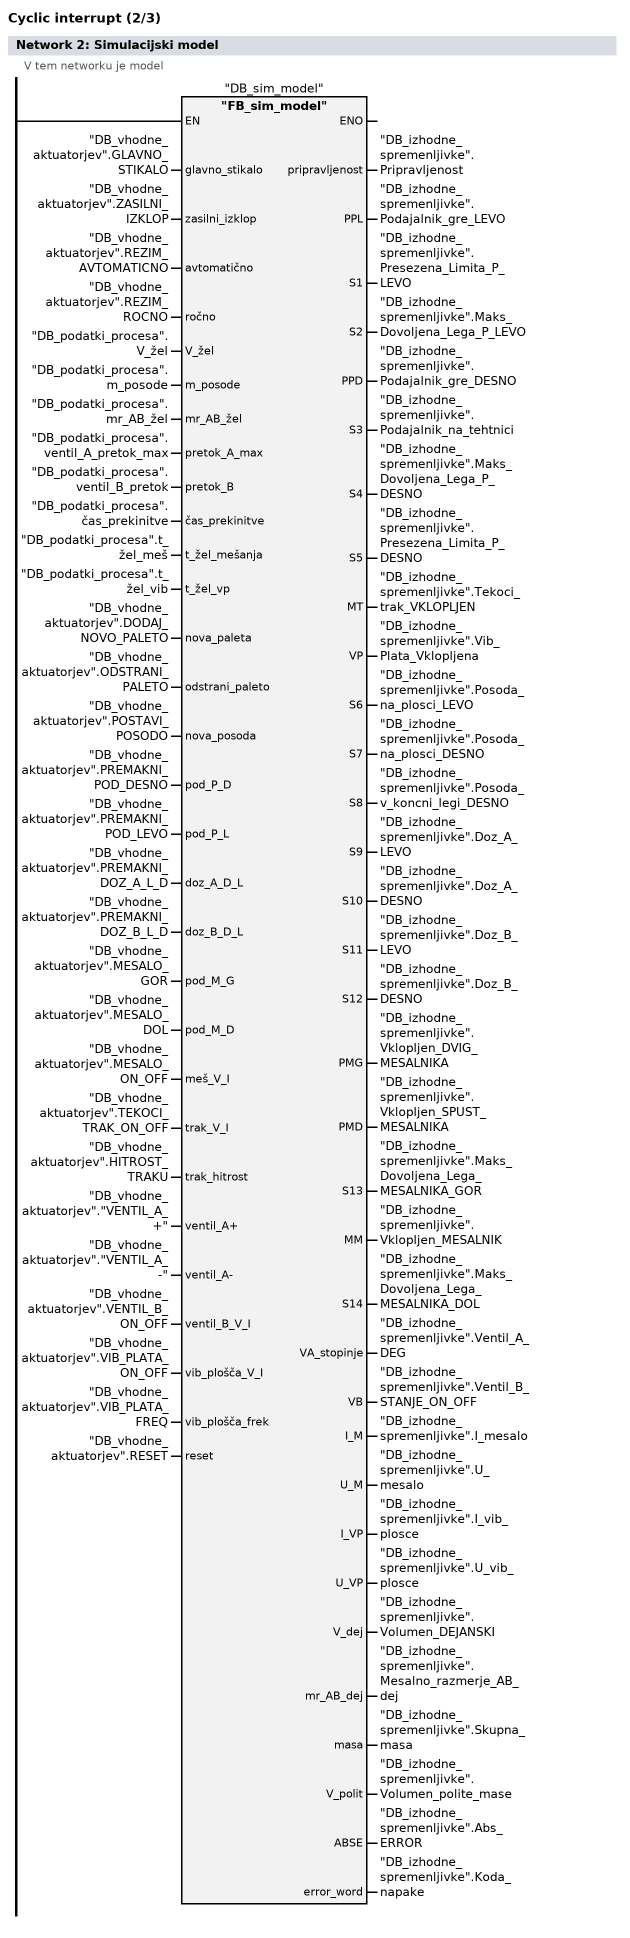
   RUNG wire#powerrail
      "DB_sim_model"(glavno_stikalo := "DB_vhodne_aktuatorjev".GLAVNO_STIKALO, zasilni_izklop := "DB_vhodne_aktuatorjev".ZASILNI_IZKLOP, avtomatično := "DB_vhodne_aktuatorjev".REZIM_AVTOMATICNO, ročno := "DB_vhodne_aktuatorjev".REZIM_ROCNO, V_žel := "DB_podatki_procesa".V_žel, m_posode := "DB_podatki_procesa".m_posode, mr_AB_žel := "DB_podatki_procesa".mr_AB_žel, pretok_A_max := "DB_podatki_procesa".ventil_A_pretok_max, pretok_B := "DB_podatki_procesa".ventil_B_pretok, čas_prekinitve := "DB_podatki_procesa".čas_prekinitve, t_žel_mešanja := "DB_podatki_procesa".t_žel_meš, t_žel_vp := "DB_podatki_procesa".t_žel_vib, nova_paleta := "DB_vhodne_aktuatorjev".DODAJ_NOVO_PALETO, odstrani_paleto := "DB_vhodne_aktuatorjev".ODSTRANI_PALETO, nova_posoda := "DB_vhodne_aktuatorjev".POSTAVI_POSODO, pod_P_D := "DB_vhodne_aktuatorjev".PREMAKNI_POD_DESNO, pod_P_L := "DB_vhodne_aktuatorjev".PREMAKNI_POD_LEVO, doz_A_D_L := "DB_vhodne_aktuatorjev".PREMAKNI_DOZ_A_L_D, doz_B_D_L := "DB_vhodne_aktuatorjev".PREMAKNI_DOZ_B_L_D, pod_M_G := "DB_vhodne_aktuatorjev".MESALO_GOR, pod_M_D := "DB_vhodne_aktuatorjev".MESALO_DOL, meš_V_I := "DB_vhodne_aktuatorjev".MESALO_ON_OFF, trak_V_I := "DB_vhodne_aktuatorjev".TEKOCI_TRAK_ON_OFF, trak_hitrost := "DB_vhodne_aktuatorjev".HITROST_TRAKU, "ventil_A+" := "DB_vhodne_aktuatorjev"."VENTIL_A_+", "ventil_A-" := "DB_vhodne_aktuatorjev"."VENTIL_A_-", ventil_B_V_I := "DB_vhodne_aktuatorjev".VENTIL_B_ON_OFF, vib_plošča_V_I := "DB_vhodne_aktuatorjev".VIB_PLATA_ON_OFF, vib_plošča_frek := "DB_vhodne_aktuatorjev".VIB_PLATA_FREQ, reset := "DB_vhodne_aktuatorjev".RESET, pripravljenost => "DB_izhodne_spremenljivke".Pripravljenost, PPL => "DB_izhodne_spremenljivke".Podajalnik_gre_LEVO, S1 => "DB_izhodne_spremenljivke".Presezena_Limita_P_LEVO, S2 => "DB_izhodne_spremenljivke".Maks_Dovoljena_Lega_P_LEVO, PPD => "DB_izhodne_spremenljivke".Podajalnik_gre_DESNO, S3 => "DB_izhodne_spremenljivke".Podajalnik_na_tehtnici, S4 => "DB_izhodne_spremenljivke".Maks_Dovoljena_Lega_P_DESNO, S5 => "DB_izhodne_spremenljivke".Presezena_Limita_P_DESNO, MT => "DB_izhodne_spremenljivke".Tekoci_trak_VKLOPLJEN, VP => "DB_izhodne_spremenljivke".Vib_Plata_Vklopljena, S6 => "DB_izhodne_spremenljivke".Posoda_na_plosci_LEVO, S7 => "DB_izhodne_spremenljivke".Posoda_na_plosci_DESNO, S8 => "DB_izhodne_spremenljivke".Posoda_v_koncni_legi_DESNO, S9 => "DB_izhodne_spremenljivke".Doz_A_LEVO, S10 => "DB_izhodne_spremenljivke".Doz_A_DESNO, S11 => "DB_izhodne_spremenljivke".Doz_B_LEVO, S12 => "DB_izhodne_spremenljivke".Doz_B_DESNO, PMG => "DB_izhodne_spremenljivke".Vklopljen_DVIG_MESALNIKA, PMD => "DB_izhodne_spremenljivke".Vklopljen_SPUST_MESALNIKA, S13 => "DB_izhodne_spremenljivke".Maks_Dovoljena_Lega_MESALNIKA_GOR, MM => "DB_izhodne_spremenljivke".Vklopljen_MESALNIK, S14 => "DB_izhodne_spremenljivke".Maks_Dovoljena_Lega_MESALNIKA_DOL, VA_stopinje => "DB_izhodne_spremenljivke".Ventil_A_DEG, VB => "DB_izhodne_spremenljivke".Ventil_B_STANJE_ON_OFF, I_M => "DB_izhodne_spremenljivke".I_mesalo, U_M => "DB_izhodne_spremenljivke".U_mesalo, I_VP => "DB_izhodne_spremenljivke".I_vib_plosce, U_VP => "DB_izhodne_spremenljivke".U_vib_plosce, V_dej => "DB_izhodne_spremenljivke".Volumen_DEJANSKI, mr_AB_dej => "DB_izhodne_spremenljivke".Mesalno_razmerje_AB_dej, masa => "DB_izhodne_spremenljivke".Skupna_masa, V_polit => "DB_izhodne_spremenljivke".Volumen_polite_mase, ABSE => "DB_izhodne_spremenljivke".Abs_ERROR, error_word => "DB_izhodne_spremenljivke".Koda_napake)
   END_RUNG
   // the same network as SCL:
   "DB_sim_model"(glavno_stikalo := "DB_vhodne_aktuatorjev".GLAVNO_STIKALO,   // "FB_sim_model"
                  zasilni_izklop := "DB_vhodne_aktuatorjev".ZASILNI_IZKLOP,
                  avtomatično := "DB_vhodne_aktuatorjev".REZIM_AVTOMATICNO,
                  ročno := "DB_vhodne_aktuatorjev".REZIM_ROCNO,
                  V_žel := "DB_podatki_procesa".V_žel,
                  m_posode := "DB_podatki_procesa".m_posode,
                  mr_AB_žel := "DB_podatki_procesa".mr_AB_žel,
                  pretok_A_max := "DB_podatki_procesa".ventil_A_pretok_max,
                  pretok_B := "DB_podatki_procesa".ventil_B_pretok,
                  čas_prekinitve := "DB_podatki_procesa".čas_prekinitve,
                  t_žel_mešanja := "DB_podatki_procesa".t_žel_meš,
                  t_žel_vp := "DB_podatki_procesa".t_žel_vib,
                  nova_paleta := "DB_vhodne_aktuatorjev".DODAJ_NOVO_PALETO,
                  odstrani_paleto := "DB_vhodne_aktuatorjev".ODSTRANI_PALETO,
                  nova_posoda := "DB_vhodne_aktuatorjev".POSTAVI_POSODO,
                  pod_P_D := "DB_vhodne_aktuatorjev".PREMAKNI_POD_DESNO,
                  pod_P_L := "DB_vhodne_aktuatorjev".PREMAKNI_POD_LEVO,
                  doz_A_D_L := "DB_vhodne_aktuatorjev".PREMAKNI_DOZ_A_L_D,
                  doz_B_D_L := "DB_vhodne_aktuatorjev".PREMAKNI_DOZ_B_L_D,
                  pod_M_G := "DB_vhodne_aktuatorjev".MESALO_GOR,
                  pod_M_D := "DB_vhodne_aktuatorjev".MESALO_DOL,
                  meš_V_I := "DB_vhodne_aktuatorjev".MESALO_ON_OFF,
                  trak_V_I := "DB_vhodne_aktuatorjev".TEKOCI_TRAK_ON_OFF,
                  trak_hitrost := "DB_vhodne_aktuatorjev".HITROST_TRAKU,
                  "ventil_A+" := "DB_vhodne_aktuatorjev"."VENTIL_A_+",
                  "ventil_A-" := "DB_vhodne_aktuatorjev"."VENTIL_A_-",
                  ventil_B_V_I := "DB_vhodne_aktuatorjev".VENTIL_B_ON_OFF,
                  vib_plošča_V_I := "DB_vhodne_aktuatorjev".VIB_PLATA_ON_OFF,
                  vib_plošča_frek := "DB_vhodne_aktuatorjev".VIB_PLATA_FREQ,
                  reset := "DB_vhodne_aktuatorjev".RESET,
                  pripravljenost => "DB_izhodne_spremenljivke".Pripravljenost,
                  PPL => "DB_izhodne_spremenljivke".Podajalnik_gre_LEVO,
                  S1 => "DB_izhodne_spremenljivke".Presezena_Limita_P_LEVO,
                  S2 => "DB_izhodne_spremenljivke".Maks_Dovoljena_Lega_P_LEVO,
                  PPD => "DB_izhodne_spremenljivke".Podajalnik_gre_DESNO,
                  S3 => "DB_izhodne_spremenljivke".Podajalnik_na_tehtnici,
                  S4 => "DB_izhodne_spremenljivke".Maks_Dovoljena_Lega_P_DESNO,
                  S5 => "DB_izhodne_spremenljivke".Presezena_Limita_P_DESNO,
                  MT => "DB_izhodne_spremenljivke".Tekoci_trak_VKLOPLJEN,
                  VP => "DB_izhodne_spremenljivke".Vib_Plata_Vklopljena,
                  S6 => "DB_izhodne_spremenljivke".Posoda_na_plosci_LEVO,
                  S7 => "DB_izhodne_spremenljivke".Posoda_na_plosci_DESNO,
                  S8 => "DB_izhodne_spremenljivke".Posoda_v_koncni_legi_DESNO,
                  S9 => "DB_izhodne_spremenljivke".Doz_A_LEVO,
                  S10 => "DB_izhodne_spremenljivke".Doz_A_DESNO,
                  S11 => "DB_izhodne_spremenljivke".Doz_B_LEVO,
                  S12 => "DB_izhodne_spremenljivke".Doz_B_DESNO,
                  PMG => "DB_izhodne_spremenljivke".Vklopljen_DVIG_MESALNIKA,
                  PMD => "DB_izhodne_spremenljivke".Vklopljen_SPUST_MESALNIKA,
                  S13 => "DB_izhodne_spremenljivke".Maks_Dovoljena_Lega_MESALNIKA_GOR,
                  MM => "DB_izhodne_spremenljivke".Vklopljen_MESALNIK,
                  S14 => "DB_izhodne_spremenljivke".Maks_Dovoljena_Lega_MESALNIKA_DOL,
                  VA_stopinje => "DB_izhodne_spremenljivke".Ventil_A_DEG,
                  VB => "DB_izhodne_spremenljivke".Ventil_B_STANJE_ON_OFF,
                  I_M => "DB_izhodne_spremenljivke".I_mesalo,
                  U_M => "DB_izhodne_spremenljivke".U_mesalo,
                  I_VP => "DB_izhodne_spremenljivke".I_vib_plosce,
                  U_VP => "DB_izhodne_spremenljivke".U_vib_plosce,
                  V_dej => "DB_izhodne_spremenljivke".Volumen_DEJANSKI,
                  mr_AB_dej => "DB_izhodne_spremenljivke".Mesalno_razmerje_AB_dej,
                  masa => "DB_izhodne_spremenljivke".Skupna_masa,
                  V_polit => "DB_izhodne_spremenljivke".Volumen_polite_mase,
                  ABSE => "DB_izhodne_spremenljivke".Abs_ERROR,
                  error_word => "DB_izhodne_spremenljivke".Koda_napake);
END_REGION

REGION Network 3
   // FB za izracun energije
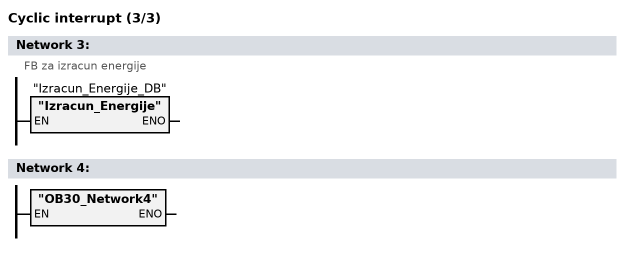
   RUNG wire#powerrail
      "Izracun_Energije_DB"()
   END_RUNG
   // the same network as SCL:
   "Izracun_Energije_DB"();   // "Izracun_Energije"
END_REGION

REGION Network 4
   RUNG wire#powerrail
      "OB30_Network4"()
   END_RUNG
   // the same network as SCL:
   "OB30_Network4"();
END_REGION
END_ORGANIZATION_BLOCK

ORGANIZATION_BLOCK "Startup"   // OB100, LAD, Startup
TITLE = "Complete Restart"
{ S7_Optimized_Access := 'TRUE' }
VERSION : 0.1
   VAR_INPUT
      LostRetentive : Bool;   // True if retentive data are lost
      LostRTC : Bool;   // True if date and time are lost
   END_VAR
BEGIN

REGION Network 1: Klic funkcije FC_init
   // Pogoj za klic FC_init je vezan na remanentno spremenljivko init_pogoj
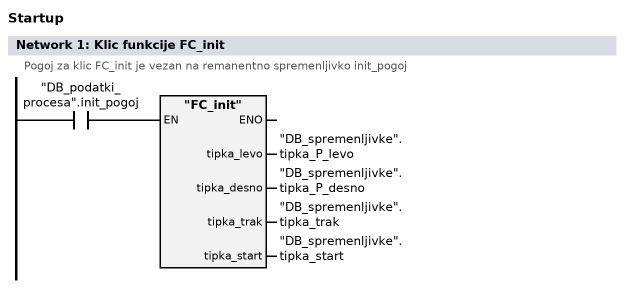
   RUNG wire#powerrail
      Contact( "DB_podatki_procesa".init_pogoj )
      "FC_init"(tipka_levo => "DB_spremenljivke".tipka_P_levo, tipka_desno => "DB_spremenljivke".tipka_P_desno, tipka_trak => "DB_spremenljivke".tipka_trak, tipka_start => "DB_spremenljivke".tipka_start)
   END_RUNG
   // the same network as SCL:
   IF "DB_podatki_procesa".init_pogoj THEN
       "FC_init"(tipka_levo => "DB_spremenljivke".tipka_P_levo,
                 tipka_desno => "DB_spremenljivke".tipka_P_desno,
                 tipka_trak => "DB_spremenljivke".tipka_trak,
                 tipka_start => "DB_spremenljivke".tipka_start);
   END_IF;
END_REGION
END_ORGANIZATION_BLOCK

(* ===== HMI "HMI_RT_1" =====
system functions are stored by id; their names below are inferred from use
connection "HMI_Connection_1": ETHERNET, S7_1200_OMS

HMI tags "Default tag table"
   "FB_sim_model_DB_stevec_prekinitev" : Int = PLC DB_sim_model.stevec_prekinitev, 100 ms
   "FB_sim_model_DB_nova_plastenka_visible" : Bool = PLC DB_sim_model.nova_posoda_visible, 100 ms
   "FB_sim_model_DB_nova_plastenka_trak_visible" : Bool = PLC DB_sim_model.nova_posoda_trak_visible, 100 ms
   "FB_sim_model_DB_stevec_prekinitev_trak" : Int = PLC DB_sim_model.stevec_prekinitev_trak, 100 ms
   "FB_sim_model_DB_trak_indikacija" : Bool = PLC DB_sim_model.MT, 100 ms
   "FB_sim_model_DB_ventil_stopinje" : Real = PLC DB_sim_model.VA_stopinje, 100 ms
   "FB_sim_model_DB_masa" : Real = PLC DB_sim_model.masa, 100 ms
   "FB_sim_model_DB_volumen_covidol" : Real = PLC DB_sim_model.volumen_AB_tehtnica, 100 ms
   "FB_sim_model_DB_stevec_plastenk" : Int = PLC DB_sim_model.stevec_posod, 100 ms
   "FB_sim_model_DB_plastenka_1_polna" : Real = PLC DB_sim_model.posoda_1, 100 ms
   "FB_sim_model_DB_plastenka_2_polna" : Real = PLC DB_sim_model.posoda_2, 100 ms
   "FB_sim_model_DB_plastenka_3_polna" : Real = PLC DB_sim_model.posoda_3, 100 ms
   "FB_sim_model_DB_plastenka_4_polna" : Real = PLC DB_sim_model.posoda_4, 100 ms
   "FB_sim_model_DB_plastenka_5_polna" : Real = PLC DB_sim_model.posoda_5, 100 ms
   "FB_sim_model_DB_plastenka_6_polna" : Real = PLC DB_sim_model.posoda_6, 100 ms
   "FB_sim_model_DB_volumen_covidol_trak" : Real = PLC DB_sim_model.volumen_v_posodi_trak, 100 ms
   "FB_sim_model_DB_nova_skatla_visible" : Bool = PLC DB_sim_model.nova_paleta_visible, 100 ms
   "FB_sim_model_DB_V_plastenke_max" : Real = PLC DB_sim_model.V_posode_max, 100 ms
   "FB_sim_model_DB_podajalnik_levo_error" : Bool = PLC DB_sim_model.S1, 100 ms
   "FB_sim_model_DB_podajalnik_tehtnica_indikacija" : Bool = PLC DB_sim_model.S3, 100 ms
   "FB_sim_model_DB_podajalnik_desno_lim_indikacija" : Bool = PLC DB_sim_model.S4, 100 ms
   "FB_sim_model_DB_podajalnik_desno_error" : Bool = PLC DB_sim_model.S5, 100 ms
   "FB_sim_model_DB_komora_levo_indikacija" : Bool = PLC DB_sim_model.S6, 100 ms
   "FB_sim_model_DB_komora_desno_indikacija" : Bool = PLC DB_sim_model.S7, 100 ms
   "FB_sim_model_DB_trak_desno_indikacija" : Bool = PLC DB_sim_model.S8, 100 ms
   "DB_sim_model_podajalnik_A_desno_lim_indikacija" : Bool = PLC DB_sim_model.S10, 100 ms
   "DB_sim_model_podajalnik_A_levo_lim_indikacija" : Bool = PLC DB_sim_model.S9, 100 ms
   "DB_sim_model_podajalnik_B_levo_lim_indikacija" : Bool = PLC DB_sim_model.S11, 100 ms
   "DB_sim_model_podajalnik_B_desno_lim_indikacija" : Bool = PLC DB_sim_model.S12, 100 ms
   "DB_sim_model_meš1_vis" : Bool = PLC DB_sim_model.meš1_vis, 100 ms
   "DB_sim_model_meš2_vis" : Bool = PLC DB_sim_model.meš2_vis, 100 ms
   "DB_sim_model_meš3_vis" : Bool = PLC DB_sim_model.meš3_vis, 100 ms
   "DB_sim_model_meš4_vis" : Bool = PLC DB_sim_model.meš4_vis, 100 ms
   "DB_sim_model_stev_prek_GD" : Int = PLC DB_sim_model.stev_prek_GD, 100 ms
   "DB_sim_model_podajalnik_gor_lim_indikacija" : Bool = PLC DB_sim_model.S13, 100 ms
   "DB_sim_model_podajalnik_dol_lim_indikacija" : Bool = PLC DB_sim_model.S14, 100 ms
   "DB_sim_model_podajalnik_dol_indikacija" : Bool = PLC DB_sim_model.PMD, 100 ms
   "DB_sim_model_podajalnik_gor_indikacija" : Bool = PLC DB_sim_model.PMG, 100 ms
   "DB_spremenljivke_reset" : Bool = PLC DB_spremenljivke.reset, 100 ms
   "DB_spremenljivke_glavno_stikalo" : Bool = PLC DB_spremenljivke.glavno_stikalo, 100 ms
   "DB_spremenljivke_zasilni_izklop" : Bool = PLC DB_spremenljivke.zasilni_izklop, 100 ms
   "DB_sim_model_ventil_B_indikacija" : Bool = PLC DB_sim_model.VB, 100 ms
   "DB_sim_model_pod_P_levo_vklop_indikacija" : Bool = PLC DB_sim_model.PPL, 100 ms
   "DB_sim_model_pod_P_desno_vklop_indikacija" : Bool = PLC DB_sim_model.PPD, 100 ms
   "DB_sim_model_pod_P_levo_lim_indikacija" : Bool = PLC DB_sim_model.S2, 100 ms
   "DB_sim_model_v_plošča_vklop_indikacija" : Bool = PLC DB_sim_model.VP, 100 ms
   "DB_sim_model_vp_visible" : Bool = PLC DB_sim_model.vp_visible, 100 ms
   "DB_sim_model_mešalo_vklop_indikacija" : Bool = PLC DB_sim_model.MM, 100 ms
   "DB_sim_model_pod_B_pos" : Int = PLC DB_sim_model.pod_B_pos, 100 ms
   "DB_sim_model_pod_A_pos" : Int = PLC DB_sim_model.pod_A_pos, 100 ms
   "DB_spremenljivke_tipka_P_levo" : Bool = PLC DB_spremenljivke.tipka_P_levo, 100 ms
   "DB_spremenljivke_tipka_P_desno" : Bool = PLC DB_spremenljivke.tipka_P_desno, 100 ms
   "DB_spremenljivke_tipka_trak" : Bool = PLC DB_spremenljivke.tipka_trak, 100 ms
   "DB_spremenljivke_dodaj_novo_paleto" : Bool = PLC DB_spremenljivke.dodaj_novo_paleto, 1 s
   "DB_spremenljivke_odstrani_paleto" : Bool = PLC DB_spremenljivke.odstrani_paleto, 1 s
   "DB_spremenljivke_postavi_novo_posodo" : Bool = PLC DB_spremenljivke.postavi_novo_posodo, 1 s
   "DB_spremenljivke_premik_dozirnika_A_levo_desno" : Bool = PLC DB_spremenljivke.premik_dozirnika_A_levo_desno, 1 s
   "DB_spremenljivke_premik_dozirnika_B_levo_desno" : Bool = PLC DB_spremenljivke.premik_dozirnika_B_levo_desno, 1 s
   "DB_spremenljivke_pod_mesalo_dol" : Bool = PLC DB_spremenljivke.pod_mesalo_dol, 1 s
   "DB_spremenljivke_pod_mesalo_gor" : Bool = PLC DB_spremenljivke.pod_mesalo_gor, 1 s
   "DB_spremenljivke_ventil_A+" : Bool = PLC DB_spremenljivke.ventil_A+, 1 s
   "DB_spremenljivke_ventil_A-" : Bool = PLC DB_spremenljivke.ventil_A-, 1 s
   "DB_spremenljivke_vklop_izklop_ventila_B" : Bool = PLC DB_spremenljivke.vklop_izklop_ventila_B, 1 s
   "DB_spremenljivke_vklopi_izklopi_mesalo" : Bool = PLC DB_spremenljivke.vklopi_izklopi_mesalo, 1 s
   "DB_spremenljivke_vklopi_izklopi_trak" : Bool = PLC DB_spremenljivke.vklopi_izklopi_trak, 1 s
   "DB_spremenljivke_vklop_izklop_VIB_plosce" : Bool = PLC DB_spremenljivke.vklop_izklop_VIB_plosce, 1 s
   "DB_podatki_procesa_V_žel" : Real = PLC DB_podatki_procesa.V_žel, 1 s
   "DB_izhodne_spremenljivke_Volumen_DEJANSKI" : Real = PLC DB_izhodne_spremenljivke.Volumen_DEJANSKI, 1 s
   "DB_izhodne_spremenljivke_Mesalno_razmerje_AB_dej" : Real = PLC DB_izhodne_spremenljivke.Mesalno_razmerje_AB_dej, 1 s
   "DB_izhodne_spremenljivke_Volumen_polite_mase" : Real = PLC DB_izhodne_spremenljivke.Volumen_polite_mase, 1 s
   "Izracun_Energije_DB_Akumulirana_energija_vib_plosce" : Real = PLC Izracun_Energije_DB.Akumulirana_energija_vib_plosce, 1 s
   "Izracun_Energije_DB_Akumulirana_energija_mesala" : Real = PLC Izracun_Energije_DB.Akumulirana_energija_mesala, 1 s
   "DB_izhodne_spremenljivke_Koda_napake" : Word = PLC DB_izhodne_spremenljivke.Koda_napake, 1 s
   "DB_vhodne_aktuatorjev_REZIM_ROCNO" : Bool = PLC DB_vhodne_aktuatorjev.REZIM_ROCNO, 1 s
   "DB_vhodne_aktuatorjev_REZIM_AVTOMATICNO" : Bool = PLC DB_vhodne_aktuatorjev.REZIM_AVTOMATICNO, 1 s
   "DB_spremenljivke_rezim_avtomaticno" : Bool = PLC DB_spremenljivke.rezim_avtomaticno, 1 s
   "DB_izhodne_spremenljivke_Pripravljenost" : Bool = PLC DB_izhodne_spremenljivke.Pripravljenost, 1 s
   "DB_spremenljivke_tipka_start" : Bool = PLC DB_spremenljivke.tipka_start, 1 s
   "DB_spremenljivke_tipka_stop" : Bool = PLC DB_spremenljivke.tipka_stop, 1 s

screen "Root screen" 800x480, template "Template_1"
   GraphicView "Graphic view_7" at 103,193 size 17x16; Picture "Graphic_21"
   GraphicView "Graphic view_4" at 53,187 size 65x22; Picture "Graphic_15"
   GraphicView "Graphic view_1" at 103,174 size 17x16; Picture "Graphic_21"
   GraphicView "Graphic view_2" at 53,168 size 65x22; Picture "Graphic_15"
   GraphicView "Graphic view_13" at 140,85 size 26x88; Picture "Graphic_48"
      Visibility <- "DB_sim_model_meš1_vis"
   GraphicView "Graphic view_6" at 140,85 size 26x88; Picture "Graphic_49"
      Visibility <- "DB_sim_model_meš4_vis"
   GraphicView "Graphic view_9" at 140,85 size 26x88; Picture "Graphic_46"
      Visibility <- "DB_sim_model_meš3_vis"
   GraphicView "Graphic view_10" at 140,85 size 26x88; Picture "Graphic_47"
      Visibility <- "DB_sim_model_meš2_vis"
   GraphicView "Graphic view_3" at 5,232 size 557x128; Picture "Graphic_60"
   Bar "Bar_1" at 47,220 size 30x38; MinimumValue 0; MaximumValue 520
      HorizontalMovement <- "FB_sim_model_DB_stevec_prekinitev"
      Visibility <- "FB_sim_model_DB_nova_plastenka_visible"
      ProcessValue <- "FB_sim_model_DB_volumen_covidol"
      MaximumValue <- "FB_sim_model_DB_V_plastenke_max"
   Group "Group_8" at 140,85 size 26x88; Picture "Graphic_48"
      VerticalMovement <- "DB_sim_model_stev_prek_GD"
   Bar "Bar_8" at 648,298 size 30x38; MinimumValue 0; MaximumValue 520
      Visibility <- "FB_sim_model_DB_stevec_plastenk"
      MaximumValue <- "FB_sim_model_DB_V_plastenke_max"
      ProcessValue <- "FB_sim_model_DB_plastenka_6_polna"
   Bar "Bar_7" at 615,298 size 30x38; MinimumValue 0; MaximumValue 520
      Visibility <- "FB_sim_model_DB_stevec_plastenk"
      MaximumValue <- "FB_sim_model_DB_V_plastenke_max"
      ProcessValue <- "FB_sim_model_DB_plastenka_5_polna"
   Bar "Bar_6" at 582,298 size 30x38; MinimumValue 0; MaximumValue 520
      Visibility <- "FB_sim_model_DB_stevec_plastenk"
      MaximumValue <- "FB_sim_model_DB_V_plastenke_max"
      ProcessValue <- "FB_sim_model_DB_plastenka_4_polna"
   Bar "Bar_2" at 186,221 size 30x38; MinimumValue 0; MaximumValue 520
      Visibility <- "FB_sim_model_DB_nova_plastenka_trak_visible"
      HorizontalMovement <- "FB_sim_model_DB_stevec_prekinitev_trak"
      ProcessValue <- "FB_sim_model_DB_volumen_covidol_trak"
      MaximumValue <- "FB_sim_model_DB_V_plastenke_max"
   IOField "I/O field_2" at 124,284 size 51x18; FormatPattern 99999; Unit  g
      ProcessValue <- "FB_sim_model_DB_masa"
   Rectangle "Rectangle_1" at 15,235 size 33x13
      HorizontalMovement <- "FB_sim_model_DB_stevec_prekinitev"
   GraphicIOField "PlotLight_Square_N_Mono" at 65,288 size 22x12; PictureOn "PilotLight_Square_N_On_mono"; PictureOff "PilotLight_Square_N_Off_mono"
      ProcessValue <- "DB_sim_model_pod_P_levo_lim_indikacija"
   GraphicIOField "PlotLight_Square_N_Mono_1" at 140,268 size 22x12; PictureOff "PilotLight_Square_N_Off_mono"; PictureOn "PilotLight_Square_N_On_mono"
      ProcessValue <- "FB_sim_model_DB_podajalnik_tehtnica_indikacija"
   GraphicIOField "PlotLight_Square_N_Mono_2" at 185,287 size 22x12; PictureOff "PilotLight_Square_N_Off_mono"; PictureOn "PilotLight_Square_N_On_mono"
      ProcessValue <- "FB_sim_model_DB_podajalnik_desno_lim_indikacija"
   GraphicIOField "PlotLight_Square_N_Mono_4" at 206,287 size 22x12; PictureOff "PilotLight_Square_N_Off_mono"; PictureOn "PilotLight_Square_R_On_256c"
      ProcessValue <- "FB_sim_model_DB_podajalnik_desno_error"
   GraphicIOField "PlotLight_Square_N_Mono_3" at 45,288 size 22x12; PictureOn "PilotLight_Square_R_On_256c"; PictureOff "PilotLight_Square_N_Off_mono"
      ProcessValue <- "FB_sim_model_DB_podajalnik_levo_error"
   GraphicIOField "PlotLight_Square_N_Mono_6" at 533,287 size 22x12; PictureOff "PilotLight_Square_N_Off_mono"; PictureOn "PilotLight_Square_N_On_mono"
      ProcessValue <- "FB_sim_model_DB_trak_desno_indikacija"
   GraphicIOField "PlotLight_Square_N_Mono_7" at 225,287 size 22x12; PictureOn "PilotLight_Square_G_On_256c"; PictureOff "PilotLight_Square_N_Off_mono"
      ProcessValue <- "FB_sim_model_DB_trak_indikacija"
   TextField "Text field_2" at 49,287 size 18x14; Text 'S1'
   TextField "Text field_3" at 69,287 size 18x14; Text 'S2'
   TextField "Text field_4" at 143,267 size 17x14; Text 'S3'
   TextField "Text field_5" at 187,286 size 17x14; Text 'S4'
   TextField "Text field_6" at 208,286 size 17x14; Text 'S5'
   TextField "Text field_7" at 536,286 size 17x14; Text 'S8'
   GraphicIOField "PlotLight_Square_N_Mono_8" at 95,288 size 22x12; PictureOn "PilotLight_Square_G_On_256c"; PictureOff "PilotLight_Square_N_Off_mono"
      ProcessValue <- "DB_sim_model_pod_P_desno_vklop_indikacija"
   TextField "Text field_9" at 94,288 size 23x11; Text 'PPD'
   TextField "Text field_8" at 227,286 size 19x14; Text 'MT'
   Switch "Rotary_RG" at 13,391 size 53x49; CaptionText 'Switch'; TextOff '0'; TextOn '1'; PictureOff "Rotary_RG_Off_256c"; PictureOn "Rotary_RG_On_256c"
      ProcessValue <- "DB_spremenljivke_glavno_stikalo"
   Switch "Pushbutton_Emergency" at 77,391 size 53x49; CaptionText 'Switch'; TextOff '0'; TextOn '1'; PictureOff "Pushbutton_Emergency_Off_256c"; PictureOn "Pushbutton_Emergency_On_256c"
      ProcessValue <- "DB_spremenljivke_zasilni_izklop"
   GraphicIOField "PlotLight_Square_N_Mono_5" at 273,287 size 22x12; PictureOff "PilotLight_Square_N_Off_mono"; PictureOn "PilotLight_Square_N_On_mono"
      ProcessValue <- "FB_sim_model_DB_komora_levo_indikacija"
   TextField "Text field_13" at 276,286 size 17x14; Text 'S6'
   GraphicIOField "PlotLight_Square_N_Mono_10" at 461,287 size 22x12; PictureOff "PilotLight_Square_N_Off_mono"; PictureOn "PilotLight_Square_N_On_mono"
      ProcessValue <- "FB_sim_model_DB_komora_desno_indikacija"
   TextField "Text field_14" at 464,286 size 17x14; Text 'S7'
   GraphicIOField "PlotLight_Square_N_Mono_9" at 16,288 size 22x12; PictureOff "PilotLight_Square_N_Off_mono"; PictureOn "PilotLight_Square_G_On_256c"
      ProcessValue <- "DB_sim_model_pod_P_levo_vklop_indikacija"
   TextField "Text field_10" at 16,287 size 24x14; Text 'PPL'
   Group "Group_6" at 53,187 size 67x22; Picture "Graphic_21"
      HorizontalMovement <- "DB_sim_model_pod_B_pos"
   Group "Group_7" at 53,168 size 67x22; Picture "Graphic_21"
      HorizontalMovement <- "DB_sim_model_pod_A_pos"
   GraphicIOField "PlotLight_Square_N_Mono_11" at 80,174 size 22x12; PictureOff "PilotLight_Square_N_Off_mono"; PictureOn "PilotLight_Square_N_On_mono"
      ProcessValue <- "DB_sim_model_podajalnik_A_desno_lim_indikacija"
   GraphicIOField "PlotLight_Square_N_Mono_14" at 11,174 size 22x12; PictureOff "PilotLight_Square_N_Off_mono"; PictureOn "PilotLight_Square_N_On_mono"
      ProcessValue <- "DB_sim_model_podajalnik_A_levo_lim_indikacija"
   GraphicIOField "PlotLight_Square_N_Mono_15" at 79,192 size 22x12; PictureOff "PilotLight_Square_N_Off_mono"; PictureOn "PilotLight_Square_N_On_mono"
      ProcessValue <- "DB_sim_model_podajalnik_B_desno_lim_indikacija"
   GraphicIOField "PlotLight_Square_N_Mono_18" at 11,193 size 22x12; PictureOff "PilotLight_Square_N_Off_mono"; PictureOn "PilotLight_Square_N_On_mono"
      ProcessValue <- "DB_sim_model_podajalnik_B_levo_lim_indikacija"
   GraphicIOField "PlotLight_Square_N_Mono_19" at 165,87 size 22x12; PictureOff "PilotLight_Square_N_Off_mono"; PictureOn "PilotLight_Square_N_On_mono"
      ProcessValue <- "DB_sim_model_podajalnik_gor_lim_indikacija"
   GraphicIOField "PlotLight_Square_N_Mono_20" at 165,151 size 22x12; PictureOff "PilotLight_Square_N_Off_mono"; PictureOn "PilotLight_Square_N_On_mono"
      ProcessValue <- "DB_sim_model_podajalnik_dol_lim_indikacija"
   GraphicIOField "PlotLight_Square_N_Mono_21" at 165,138 size 22x12; PictureOff "PilotLight_Square_N_Off_mono"; PictureOn "PilotLight_Square_G_On_256c"
      ProcessValue <- "DB_sim_model_podajalnik_dol_indikacija"
   GraphicIOField "PlotLight_Square_N_Mono_22" at 165,100 size 22x12; PictureOff "PilotLight_Square_N_Off_mono"; PictureOn "PilotLight_Square_G_On_256c"
      ProcessValue <- "DB_sim_model_podajalnik_gor_indikacija"
   Bar "Bar_3" at 574,299 size 30x38; MinimumValue 0; MaximumValue 520
      MaximumValue <- "FB_sim_model_DB_V_plastenke_max"
      Visibility <- "FB_sim_model_DB_stevec_plastenk"
      ProcessValue <- "FB_sim_model_DB_plastenka_1_polna"
   Bar "Bar_4" at 607,299 size 30x38; MinimumValue 0; MaximumValue 520
      Visibility <- "FB_sim_model_DB_stevec_plastenk"
      MaximumValue <- "FB_sim_model_DB_V_plastenke_max"
      ProcessValue <- "FB_sim_model_DB_plastenka_2_polna"
   Bar "Bar_5" at 640,299 size 30x38; MinimumValue 0; MaximumValue 520
      Visibility <- "FB_sim_model_DB_stevec_plastenk"
      MaximumValue <- "FB_sim_model_DB_V_plastenke_max"
      ProcessValue <- "FB_sim_model_DB_plastenka_3_polna"
   Rectangle "Rectangle_5" at 565,336 size 120x14
      Visibility <- "FB_sim_model_DB_nova_skatla_visible"
   TextField "Text field_22" at 80,173 size 24x14; Text 'S10'
   TextField "Text field_27" at 14,173 size 18x14; Text 'S9'
   TextField "Text field_28" at 80,191 size 24x14; Text 'S12'
   TextField "Text field_29" at 11,192 size 24x14; Text 'S11'
   TextField "Text field_30" at 165,150 size 24x14; Text 'S14'
   TextField "Text field_31" at 165,86 size 24x14; Text 'S13'
   TextField "Text field_32" at 163,138 size 26x11; Text 'PMD'
   TextField "Text field_33" at 163,100 size 26x11; Text 'PMG'
   Rectangle "Rectangle_2" at 275,279 size 205x4
      Visibility <- "DB_sim_model_vp_visible"
   IOField "I/O field_3" at 10,101 size 35x22; FormatPattern 99
      ProcessValue <- "FB_sim_model_DB_ventil_stopinje"
   TextField "Text field_12" at 44,104 size 18x14; Text 'st.'
   TextField "Text field_40" at 8,88 size 42x14; Text 'Ventil A'
   TextField "Text field_41" at 8,126 size 42x14; Text 'Ventil B'
   GraphicIOField "PlotLight_Square_N_Mono_23" at 10,140 size 22x12; PictureOn "PilotLight_Square_N_On_mono"; PictureOff "PilotLight_Square_N_Off_mono"
      ProcessValue <- "DB_sim_model_ventil_B_indikacija"
   TextField "Text field_42" at 11,139 size 18x14; Text 'VB'
   GraphicIOField "PlotLight_Square_N_Mono_24" at 364,288 size 22x12; PictureOn "PilotLight_Square_N_On_mono"; PictureOff "PilotLight_Square_N_Off_mono"
      ProcessValue <- "DB_sim_model_v_plošča_vklop_indikacija"
   TextField "Text field_11" at 367,287 size 17x14; Text 'VP'
   GraphicIOField "PlotLight_Square_N_Mono_25" at 165,119 size 22x12; PictureOn "PilotLight_Square_N_On_mono"; PictureOff "PilotLight_Square_N_Off_mono"
      ProcessValue <- "DB_sim_model_mešalo_vklop_indikacija"
   TextField "Text field_43" at 165,118 size 22x14; Text 'MM'
   Button "Button_1" at 13,449 size 52x18; TextOff 'Reset'
      on Press: function_b14e0dd5("DB_spremenljivke_reset", 0)
   Switch "Lever_Vertical_1" at 279,397 size 50x80; CaptionText 'Switch'; TextOff '0'; TextOn '1'; PictureOff "Lever_Vertical_1_Off_256c"; PictureOn "Lever_Vertical_1_On_256c"
      ProcessValue <- "DB_spremenljivke_dodaj_novo_paleto"
   Switch "Lever_Vertical_2" at 346,395 size 50x80; CaptionText 'Switch'; TextOff '0'; TextOn '1'; PictureOff "Lever_Vertical_1_Off_256c"; PictureOn "Lever_Vertical_1_On_256c"
      ProcessValue <- "DB_spremenljivke_odstrani_paleto"
   Switch "Lever_Vertical_3" at 430,395 size 50x80; CaptionText 'Switch'; TextOff '0'; TextOn '1'; PictureOff "Lever_Vertical_1_Off_256c"; PictureOn "Lever_Vertical_1_On_256c"
      ProcessValue <- "DB_spremenljivke_postavi_novo_posodo"
   Switch "Lever_Vertical_4" at 536,400 size 50x80; CaptionText 'Switch'; TextOff '0'; TextOn '1'; PictureOff "Lever_Vertical_1_Off_256c"; PictureOn "Lever_Vertical_1_On_256c"
      ProcessValue <- "DB_spremenljivke_tipka_P_levo"
   Switch "Lever_Vertical_5" at 619,398 size 50x80; CaptionText 'Switch'; TextOff '0'; TextOn '1'; PictureOff "Lever_Vertical_1_Off_256c"; PictureOn "Lever_Vertical_1_On_256c"
      ProcessValue <- "DB_spremenljivke_tipka_P_desno"
   Switch "Lever_Vertical_6" at 702,400 size 45x78; CaptionText 'Switch'; TextOff '0'; TextOn '1'; PictureOff "Lever_Vertical_1_Off_256c"; PictureOn "Lever_Vertical_1_On_256c"
      ProcessValue <- "DB_spremenljivke_premik_dozirnika_A_levo_desno"
   Switch "Lever_Vertical_7" at 750,400 size 50x80; CaptionText 'Switch'; TextOff '0'; TextOn '1'; PictureOff "Lever_Vertical_1_Off_256c"; PictureOn "Lever_Vertical_1_On_256c"
      ProcessValue <- "DB_spremenljivke_premik_dozirnika_B_levo_desno"
   TextField "Text field_1" at 262,368 size 78x23; Text 'dod pal.'
   TextField "Text field_15" at 329,368 size 84x23; Text 'odst. pal'
   TextField "Text field_16" at 417,374 size 113x23; Text 'nova posod.'
   TextField "Text field_17" at 255,6 size 111x23; Text 'mesalo gor'
   TextField "Text field_18" at 152,4 size 108x23; Text 'mesalo_dol'
   TextField "Text field_19" at 600,372 size 103x23; Text 'pod. desno'
   TextField "Text field_20" at 677,372 size 99x23; Text 'doz A/L/D'
   TextField "Text field_21" at 519,371 size 88x23; Text 'pod. levo'
   TextField "Text field_23" at 702,349 size 98x23; Text 'doz B/L/D'
   Switch "Lever_Vertical_8" at 197,27 size 50x80; CaptionText 'Switch'; TextOff '0'; TextOn '1'; PictureOff "Lever_Vertical_1_Off_256c"; PictureOn "Lever_Vertical_1_On_256c"
      ProcessValue <- "DB_spremenljivke_pod_mesalo_dol"
   Switch "Lever_Vertical_9" at 285,27 size 50x80; CaptionText 'Switch'; TextOff '0'; TextOn '1'; PictureOff "Lever_Vertical_1_Off_256c"; PictureOn "Lever_Vertical_1_On_256c"
      ProcessValue <- "DB_spremenljivke_pod_mesalo_gor"
   Switch "Lever_Vertical_10" at 367,32 size 50x80; CaptionText 'Switch'; TextOff '0'; TextOn '1'; PictureOff "Lever_Vertical_1_Off_256c"; PictureOn "Lever_Vertical_1_On_256c"
      ProcessValue <- "DB_spremenljivke_ventil_A+"
   Switch "Lever_Vertical_11" at 433,31 size 50x80; CaptionText 'Switch'; TextOff '0'; TextOn '1'; PictureOff "Lever_Vertical_1_Off_256c"; PictureOn "Lever_Vertical_1_On_256c"
      ProcessValue <- "DB_spremenljivke_ventil_A-"
   TextField "Text field_24" at 357,10 size 78x23; Text 'vent.A+'
   TextField "Text field_25" at 425,10 size 72x23; Text 'vent.A-'
   Switch "Lever_Vertical_12" at 541,31 size 45x81; CaptionText 'Switch'; TextOff '0'; TextOn '1'; PictureOff "Lever_Vertical_1_Off_256c"; PictureOn "Lever_Vertical_1_On_256c"
      ProcessValue <- "DB_spremenljivke_vklop_izklop_ventila_B"
   Switch "Lever_Vertical_13" at 607,33 size 50x80; CaptionText 'Switch'; TextOff '0'; TextOn '1'; PictureOff "Lever_Vertical_1_Off_256c"; PictureOn "Lever_Vertical_1_On_256c"
      ProcessValue <- "DB_spremenljivke_vklopi_izklopi_mesalo"
   TextField "Text field_26" at 536,0 size 58x42; Text 'ventB _V/I'
   TextField "Text field_34" at 599,0 size 70x42; Text 'mesalo _V/I'
   Switch "Lever_Vertical_14" at 255,150 size 50x80; CaptionText 'Switch'; TextOff '0'; TextOn '1'; PictureOff "Lever_Vertical_1_Off_256c"; PictureOn "Lever_Vertical_1_On_256c"
      ProcessValue <- "DB_spremenljivke_vklopi_izklopi_trak"
   TextField "Text field_35" at 262,129 size 43x23; Text 'trak'
   Switch "Lever_Vertical_15" at 336,149 size 50x80; CaptionText 'Switch'; TextOff '0'; TextOn '1'; PictureOff "Lever_Vertical_1_Off_256c"; PictureOn "Lever_Vertical_1_On_256c"
      ProcessValue <- "DB_spremenljivke_vklop_izklop_VIB_plosce"
   TextField "Text field_36" at 324,126 size 101x23; Text 'vib. plosca'
   IOField "I/O field_1" at 16,29 size 76x27; FormatPattern s999999999.999
      ProcessValue <- "DB_podatki_procesa_V_žel"
   IOField "I/O field_5" at 717,83 size 69x34; FormatPattern s999999999.999
      ProcessValue <- "DB_izhodne_spremenljivke_Volumen_DEJANSKI"
   IOField "I/O field_6" at 715,136 size 73x30; FormatPattern s999999999.999
      ProcessValue <- "DB_izhodne_spremenljivke_Mesalno_razmerje_AB_dej"
   IOField "I/O field_7" at 711,197 size 77x32; FormatPattern s999999999.999
      ProcessValue <- "DB_izhodne_spremenljivke_Volumen_polite_mase"
   TextField "Text field_37" at 703,170 size 97x23; Text 'vol. polite'
   TextField "Text field_38" at 697,116 size 103x23; Text 'm.r AB Dej'
   TextField "Text field_39" at 725,64 size 52x23; Text 'V dej'
   TextField "Text field_44" at 0,5 size 97x23; Text 'V zel vnos'
   IOField "I/O field_4" at 417,150 size 96x32; FormatPattern s999999999.999
      ProcessValue <- "Izracun_Energije_DB_Akumulirana_energija_mesala"
   TextField "Text field_45" at 420,126 size 71x23; Text 'E. MES.'
   IOField "I/O field_8" at 524,149 size 96x32; FormatPattern s999999999.999
      ProcessValue <- "Izracun_Energije_DB_Akumulirana_energija_vib_plosce"
   TextField "Text field_46" at 534,123 size 52x23; Text 'E V.P'
   IOField "I/O field_9" at 719,28 size 67x32; FormatPattern 99999
      ProcessValue <- "DB_izhodne_spremenljivke_Koda_napake"
   TextField "Text field_47" at 727,4 size 73x23; Text 'Napaka'
   GraphicIOField "PlotLight_Round_G" at 144,366 size 19x21; PictureOn "PilotLight_Round_G_On_256c"; PictureOff "PilotLight_Round_G_Off_256c"
      ProcessValue <- "DB_vhodne_aktuatorjev_REZIM_ROCNO"
   GraphicIOField "PlotLight_Round_R" at 177,366 size 20x21; PictureOn "PilotLight_Round_R_On_256c"; PictureOff "PilotLight_Round_R_Off_256c"
      ProcessValue <- "DB_vhodne_aktuatorjev_REZIM_AVTOMATICNO"
   TextField "Text field_48" at 122,364 size 18x23; Text 'R'
   TextField "Text field_49" at 198,366 size 18x23; Text 'A'
   Button "Button_2" at 138,391 size 61x29; TextOff 'Avt.'
      on Press: function_b14e0dd5("DB_spremenljivke_rezim_avtomaticno", 0)
   Button "Button_3" at 137,420 size 62x28; TextOff 'START'
      on Press: function_b14e0dd5("DB_spremenljivke_tipka_start", 0)
   Button "Button_4" at 136,450 size 65x28; TextOff 'STOP'
      on Press: function_b14e0dd5("DB_spremenljivke_tipka_stop", 0)
   GraphicIOField "PlotLight_Round_GN" at 222,364 size 25x25; PictureOn "PilotLight_Round_GN_On_256c"; PictureOff "PilotLight_Round_GN_Off_256c"
      ProcessValue <- "DB_izhodne_spremenljivke_Pripravljenost"
   TextField "Text field_50" at 247,360 size 17x23; Text 'P'
*)